LIN {X -0.121,Y -401.497,Z 1324.427,A 0.000,B 0.000,C 90.000,E1 292.823} C_DIS
LIN {X 0.045,Y -401.770,Z 1324.423,A 0.000,B 0.000,C 90.000,E1 292.099} C_DIS
LIN {X 0.005,Y -404.574,Z 1324.396,A 0.000,B 0.000,C 90.000,E1 287.221} C_DIS
LIN {X 0.106,Y -404.760,Z 1324.394,A 0.000,B 0.000,C 90.000,E1 286.858} C_DIS
LIN {X 0.013,Y -406.044,Z 1324.365,A 0.000,B 0.000,C 90.000,E1 281.658} C_DIS
LIN {X 0.103,Y -406.134,Z 1324.363,A 0.000,B 0.000,C 90.000,E1 281.299} C_DIS
LIN {X 0.132,Y -405.657,Z 1324.334,A 0.000,B 0.000,C 90.000,E1 276.087} C_DIS
LIN {X 0.138,Y -405.595,Z 1324.332,A 0.000,B 0.000,C 90.000,E1 275.739} C_DIS
LIN {X -0.193,Y -403.547,Z 1324.305,A 0.000,B 0.000,C 90.000,E1 270.917} C_DIS
LIN {X 0.146,Y -403.030,Z 1324.301,A 0.000,B 0.000,C 90.000,E1 270.172} C_DIS
LIN {X -0.032,Y -399.006,Z 1324.272,A 0.000,B 0.000,C 90.000,E1 264.951} C_DIS
LIN {X -0.006,Y -395.117,Z 1324.254,A 0.000,B 0.000,C 90.000,E1 261.781} C_DIS
LIN {X 0.129,Y -392.916,Z 1324.241,A 0.000,B 0.000,C 90.000,E1 259.285} C_DIS
LIN {X 0.120,Y -391.854,Z 1324.237,A 0.000,B 0.000,C 90.000,E1 258.578} C_DIS
LIN {X -0.125,Y -385.723,Z 1324.211,A 0.000,B 0.000,C 90.000,E1 253.976} C_DIS
LIN {X -0.189,Y -384.951,Z 1324.207,A 0.000,B 0.000,C 90.000,E1 253.268} C_DIS
LIN {X 0.038,Y -378.101,Z 1324.183,A 0.000,B 0.000,C 90.000,E1 248.901} C_DIS
LIN {X -0.226,Y -376.344,Z 1324.175,A 0.000,B 0.000,C 90.000,E1 247.486} C_DIS
LIN {X -0.100,Y -375.834,Z 1324.173,A 0.000,B 0.000,C 90.000,E1 247.102} C_DIS
LIN {X 0.018,Y -369.070,Z 1324.150,A 0.000,B 0.000,C 90.000,E1 243.050} C_DIS
LIN {X -0.071,Y -366.221,Z 1324.138,A 0.000,B 0.000,C 90.000,E1 240.845} C_DIS
LIN {X 0.090,Y -358.817,Z 1324.113,A 0.000,B 0.000,C 90.000,E1 236.342} C_DIS
LIN {X -0.119,Y -356.008,Z 1324.101,A 0.000,B 0.000,C 90.000,E1 234.116} C_DIS
LIN {X -0.138,Y -350.728,Z 1324.083,A 0.000,B 0.000,C 90.000,E1 230.884} C_DIS
LIN {X -0.156,Y -350.742,Z 1324.083,A 0.000,B 0.000,C 90.000,E1 230.884} C_DIS
LIN {X 0.060,Y -364.108,Z 1324.069,A 0.000,B 0.000,C 90.000,E1 228.405} C_DIS
LIN {X -0.264,Y -378.946,Z 1324.056,A 0.000,B 0.000,C 90.000,E1 226.053} C_DIS
LIN {X -0.195,Y -395.284,Z 1324.043,A 0.000,B 0.000,C 90.000,E1 223.704} C_DIS
LIN {X -0.073,Y -413.058,Z 1324.030,A 0.000,B 0.000,C 90.000,E1 221.434} C_DIS
LIN {X -0.030,Y -432.976,Z 1324.018,A 0.000,B 0.000,C 90.000,E1 219.197} C_DIS
LIN {X -0.195,Y -443.092,Z 1324.012,A 0.000,B 0.000,C 90.000,E1 218.177} C_DIS
LIN {X -0.039,Y -444.761,Z 1324.010,A 0.000,B 0.000,C 90.000,E1 217.855} C_DIS
LIN {X -0.002,Y -445.959,Z 1324.009,A 0.000,B 0.000,C 90.000,E1 217.523} C_DIS
LIN {X -0.039,Y -446.904,Z 1324.007,A 0.000,B 0.000,C 90.000,E1 217.202} C_DIS
LIN {X 0.012,Y -447.701,Z 1324.005,A 0.000,B 0.000,C 90.000,E1 216.870} C_DIS
LIN {X 0.036,Y -448.929,Z 1324.001,A 0.000,B 0.000,C 90.000,E1 216.217} C_DIS
LIN {X -0.193,Y -449.875,Z 1323.998,A 0.000,B 0.000,C 90.000,E1 215.598} C_DIS
LIN {X -0.078,Y -450.866,Z 1323.992,A 0.000,B 0.000,C 90.000,E1 214.612} C_DIS
LIN {X 0.114,Y -453.547,Z 1323.978,A 0.000,B 0.000,C 90.000,E1 212.005} C_DIS
LIN {X -0.202,Y -456.066,Z 1323.965,A 0.000,B 0.000,C 90.000,E1 209.795} C_DIS
LIN {X 0.116,Y -458.841,Z 1323.953,A 0.000,B 0.000,C 90.000,E1 207.513} C_DIS
LIN {X 0.098,Y -462.041,Z 1323.941,A 0.000,B 0.000,C 90.000,E1 205.283} C_DIS
LIN {X -0.010,Y -463.926,Z 1323.933,A 0.000,B 0.000,C 90.000,E1 204.027} C_DIS
LIN {X -0.094,Y -465.699,Z 1323.927,A 0.000,B 0.000,C 90.000,E1 202.770} C_DIS
LIN {X 0.048,Y -467.836,Z 1323.918,A 0.000,B 0.000,C 90.000,E1 201.173} C_DIS
LIN {X 0.137,Y -470.708,Z 1323.906,A 0.000,B 0.000,C 90.000,E1 198.960} C_DIS
LIN {X 0.019,Y -473.212,Z 1323.895,A 0.000,B 0.000,C 90.000,E1 197.094} C_DIS
LIN {X -0.181,Y -475.587,Z 1323.885,A 0.000,B 0.000,C 90.000,E1 195.245} C_DIS
LIN {X 0.009,Y -477.937,Z 1323.874,A 0.000,B 0.000,C 90.000,E1 193.355} C_DIS
LIN {X 0.002,Y -480.638,Z 1323.862,A 0.000,B 0.000,C 90.000,E1 191.186} C_DIS
LIN {X 0.243,Y -482.542,Z 1323.854,A 0.000,B 0.000,C 90.000,E1 189.613} C_DIS
LIN {X -0.036,Y -484.416,Z 1323.845,A 0.000,B 0.000,C 90.000,E1 188.106} C_DIS
LIN {X 0.139,Y -486.155,Z 1323.837,A 0.000,B 0.000,C 90.000,E1 186.549} C_DIS
LIN {X 0.040,Y -487.423,Z 1323.830,A 0.000,B 0.000,C 90.000,E1 185.334} C_DIS
LIN {X 0.053,Y -489.054,Z 1323.819,A 0.000,B 0.000,C 90.000,E1 183.498} C_DIS
LIN {X -0.246,Y -490.104,Z 1323.811,A 0.000,B 0.000,C 90.000,E1 182.007} C_DIS
LIN {X -0.041,Y -490.805,Z 1323.803,A 0.000,B 0.000,C 90.000,E1 180.458} C_DIS
LIN {X 0.166,Y -491.124,Z 1323.794,A 0.000,B 0.000,C 90.000,E1 178.912} C_DIS
LIN {X -0.145,Y -491.170,Z 1323.791,A 0.000,B 0.000,C 90.000,E1 178.339} C_DIS
LIN {X 0.097,Y -490.879,Z 1323.782,A 0.000,B 0.000,C 90.000,E1 176.788} C_DIS
LIN {X -0.019,Y -490.174,Z 1323.776,A 0.000,B 0.000,C 90.000,E1 175.584} C_DIS
LIN {X 0.012,Y -489.462,Z 1323.770,A 0.000,B 0.000,C 90.000,E1 174.666} C_DIS
LIN {X 0.080,Y -488.430,Z 1323.765,A 0.000,B 0.000,C 90.000,E1 173.742} C_DIS
LIN {X -0.221,Y -487.716,Z 1323.762,A 0.000,B 0.000,C 90.000,E1 173.166} C_DIS
LIN {X -0.046,Y -486.853,Z 1323.759,A 0.000,B 0.000,C 90.000,E1 172.534} C_DIS
LIN {X 0.061,Y -485.258,Z 1323.753,A 0.000,B 0.000,C 90.000,E1 171.602} C_DIS
LIN {X 0.081,Y -483.312,Z 1323.748,A 0.000,B 0.000,C 90.000,E1 170.679} C_DIS
LIN {X 0.155,Y -481.094,Z 1323.743,A 0.000,B 0.000,C 90.000,E1 169.746} C_DIS
LIN {X 0.204,Y -478.140,Z 1323.738,A 0.000,B 0.000,C 90.000,E1 168.814} C_DIS
LIN {X -0.094,Y -475.795,Z 1323.735,A 0.000,B 0.000,C 90.000,E1 168.229} C_DIS
LIN {X -0.010,Y -471.370,Z 1323.729,A 0.000,B 0.000,C 90.000,E1 167.285} C_DIS
LIN {X -0.087,Y -465.612,Z 1323.724,A 0.000,B 0.000,C 90.000,E1 166.353} C_DIS
LIN {X 0.163,Y -454.836,Z 1323.714,A 0.000,B 0.000,C 90.000,E1 164.574} C_DIS
LIN {X 0.161,Y -445.144,Z 1323.705,A 0.000,B 0.000,C 90.000,E1 162.960} C_DIS
LIN {X 0.148,Y -439.297,Z 1323.699,A 0.000,B 0.000,C 90.000,E1 161.819} C_DIS
LIN {X -0.145,Y -437.494,Z 1323.696,A 0.000,B 0.000,C 90.000,E1 161.221} C_DIS
LIN {X 0.105,Y -436.906,Z 1323.694,A 0.000,B 0.000,C 90.000,E1 160.859} C_DIS
LIN {X -0.061,Y -436.819,Z 1323.692,A 0.000,B 0.000,C 90.000,E1 160.550} C_DIS
LIN {X 0.013,Y -438.051,Z 1323.690,A 0.000,B 0.000,C 90.000,E1 160.134} C_DIS
LIN {X 0.121,Y -438.069,Z 1323.690,A 0.000,B 0.000,C 90.000,E1 160.115} C_DIS
LIN {X 0.145,Y -440.213,Z 1323.688,A 0.000,B 0.000,C 90.000,E1 159.880} C_DIS
LIN {X -0.083,Y -441.492,Z 1323.688,A 0.000,B 0.000,C 90.000,E1 159.752} C_DIS
LIN {X 0.103,Y -450.346,Z 1323.683,A 0.000,B 0.000,C 90.000,E1 158.975} C_DIS
LIN {X 0.249,Y -462.852,Z 1323.678,A 0.000,B 0.000,C 90.000,E1 157.975} C_DIS
LIN {X -0.095,Y -473.715,Z 1323.673,A 0.000,B 0.000,C 90.000,E1 157.177} C_DIS
LIN {X 0.021,Y -484.245,Z 1323.668,A 0.000,B 0.000,C 90.000,E1 156.305} C_DIS
LIN {X 0.027,Y -491.350,Z 1323.665,A 0.000,B 0.000,C 90.000,E1 155.665} C_DIS
LIN {X 0.255,Y -498.290,Z 1323.661,A 0.000,B 0.000,C 90.000,E1 154.973} C_DIS
LIN {X 0.202,Y -506.494,Z 1323.657,A 0.000,B 0.000,C 90.000,E1 154.152} C_DIS
LIN {X -0.144,Y -514.176,Z 1323.652,A 0.000,B 0.000,C 90.000,E1 153.332} C_DIS
LIN {X 0.066,Y -517.855,Z 1323.649,A 0.000,B 0.000,C 90.000,E1 152.871} C_DIS
LIN {X -0.273,Y -520.234,Z 1323.648,A 0.000,B 0.000,C 90.000,E1 152.615} C_DIS
LIN {X -0.226,Y -524.431,Z 1323.645,A 0.000,B 0.000,C 90.000,E1 152.025} C_DIS
LIN {X 0.162,Y -528.939,Z 1323.641,A 0.000,B 0.000,C 90.000,E1 151.257} C_DIS
LIN {X -0.186,Y -531.948,Z 1323.637,A 0.000,B 0.000,C 90.000,E1 150.717} C_DIS
LIN {X -0.048,Y -534.414,Z 1323.634,A 0.000,B 0.000,C 90.000,E1 150.127} C_DIS
LIN {X 0.106,Y -536.377,Z 1323.631,A 0.000,B 0.000,C 90.000,E1 149.537} C_DIS
LIN {X -0.190,Y -538.148,Z 1323.628,A 0.000,B 0.000,C 90.000,E1 148.997} C_DIS
LIN {X -0.013,Y -539.691,Z 1323.625,A 0.000,B 0.000,C 90.000,E1 148.408} C_DIS
LIN {X 0.183,Y -541.656,Z 1323.620,A 0.000,B 0.000,C 90.000,E1 147.533} C_DIS
LIN {X -0.077,Y -542.760,Z 1323.617,A 0.000,B 0.000,C 90.000,E1 146.993} C_DIS
LIN {X -0.003,Y -544.135,Z 1323.612,A 0.000,B 0.000,C 90.000,E1 146.135} C_DIS
LIN {X -0.212,Y -545.265,Z 1323.607,A 0.000,B 0.000,C 90.000,E1 145.308} C_DIS
LIN {X 0.349,Y -546.179,Z 1323.603,A 0.000,B 0.000,C 90.000,E1 144.402} C_DIS
LIN {X -0.243,Y -547.175,Z 1323.596,A 0.000,B 0.000,C 90.000,E1 143.336} C_DIS
LIN {X 0.086,Y -548.739,Z 1323.585,A 0.000,B 0.000,C 90.000,E1 141.331} C_DIS
LIN {X -0.243,Y -549.253,Z 1323.582,A 0.000,B 0.000,C 90.000,E1 140.803} C_DIS
LIN {X -0.163,Y -549.755,Z 1323.581,A 0.000,B 0.000,C 90.000,E1 140.517} C_DIS
LIN {X -0.030,Y -550.405,Z 1323.579,A 0.000,B 0.000,C 90.000,E1 140.275} C_DIS
LIN {X -0.098,Y -550.908,Z 1323.579,A 0.000,B 0.000,C 90.000,E1 140.194} C_DIS
LIN {X -0.011,Y -551.251,Z 1323.579,A 0.000,B 0.000,C 90.000,E1 140.150} C_DIS
LIN {X 0.193,Y -553.747,Z 1323.578,A 0.000,B 0.000,C 90.000,E1 139.989} C_DIS
LIN {X -0.092,Y -561.011,Z 1323.577,A 0.000,B 0.000,C 90.000,E1 139.784} C_DIS
LIN {X -0.058,Y -566.314,Z 1323.576,A 0.000,B 0.000,C 90.000,E1 139.622} C_DIS
LIN {X 0.041,Y -572.536,Z 1323.574,A 0.000,B 0.000,C 90.000,E1 139.380} C_DIS
LIN {X 0.025,Y -575.274,Z 1323.574,A 0.000,B 0.000,C 90.000,E1 139.256} C_DIS
LIN {X 0.100,Y -578.139,Z 1323.573,A 0.000,B 0.000,C 90.000,E1 139.094} C_DIS
LIN {X 0.102,Y -583.931,Z 1323.571,A 0.000,B 0.000,C 90.000,E1 138.728} C_DIS
LIN {X 0.179,Y -589.629,Z 1323.569,A 0.000,B 0.000,C 90.000,E1 138.324} C_DIS
LIN {X -0.289,Y -592.300,Z 1323.568,A 0.000,B 0.000,C 90.000,E1 138.162} C_DIS
LIN {X -0.249,Y -597.402,Z 1323.565,A 0.000,B 0.000,C 90.000,E1 137.715} C_DIS
LIN {X 0.026,Y -603.693,Z 1323.562,A 0.000,B 0.000,C 90.000,E1 137.067} C_DIS
LIN {X 0.039,Y -609.589,Z 1323.558,A 0.000,B 0.000,C 90.000,E1 136.419} C_DIS
LIN {X -0.392,Y -614.960,Z 1323.554,A 0.000,B 0.000,C 90.000,E1 135.810} C_DIS
LIN {X 0.074,Y -619.928,Z 1323.551,A 0.000,B 0.000,C 90.000,E1 135.121} C_DIS
LIN {X 0.077,Y -625.397,Z 1323.547,A 0.000,B 0.000,C 90.000,E1 134.352} C_DIS
LIN {X 0.197,Y -629.756,Z 1323.543,A 0.000,B 0.000,C 90.000,E1 133.704} C_DIS
LIN {X 0.205,Y -636.392,Z 1323.537,A 0.000,B 0.000,C 90.000,E1 132.690} C_DIS
LIN {X -0.139,Y -644.193,Z 1323.530,A 0.000,B 0.000,C 90.000,E1 131.472} C_DIS
LIN {X -0.369,Y -649.561,Z 1323.526,A 0.000,B 0.000,C 90.000,E1 130.620} C_DIS
LIN {X 0.390,Y -655.307,Z 1323.520,A 0.000,B 0.000,C 90.000,E1 129.564} C_DIS
LIN {X -0.142,Y -660.174,Z 1323.515,A 0.000,B 0.000,C 90.000,E1 128.749} C_DIS
LIN {X 0.444,Y -665.225,Z 1323.510,A 0.000,B 0.000,C 90.000,E1 127.729} C_DIS
LIN {X 0.033,Y -668.149,Z 1323.506,A 0.000,B 0.000,C 90.000,E1 127.156} C_DIS
LIN {X 0.098,Y -671.391,Z 1323.502,A 0.000,B 0.000,C 90.000,E1 126.423} C_DIS
LIN {X -0.208,Y -674.346,Z 1323.498,A 0.000,B 0.000,C 90.000,E1 125.724} C_DIS
LIN {X 0.070,Y -677.016,Z 1323.494,A 0.000,B 0.000,C 90.000,E1 124.978} C_DIS
LIN {X -0.177,Y -679.417,Z 1323.490,A 0.000,B 0.000,C 90.000,E1 124.278} C_DIS
LIN {X 0.155,Y -682.105,Z 1323.485,A 0.000,B 0.000,C 90.000,E1 123.293} C_DIS
LIN {X -0.056,Y -683.932,Z 1323.481,A 0.000,B 0.000,C 90.000,E1 122.594} C_DIS
LIN {X -0.414,Y -686.028,Z 1323.476,A 0.000,B 0.000,C 90.000,E1 121.671} C_DIS
LIN {X 0.207,Y -687.810,Z 1323.471,A 0.000,B 0.000,C 90.000,E1 120.669} C_DIS
LIN {X -0.316,Y -688.916,Z 1323.467,A 0.000,B 0.000,C 90.000,E1 120.001} C_DIS
LIN {X -0.231,Y -689.846,Z 1323.463,A 0.000,B 0.000,C 90.000,E1 119.283} C_DIS
LIN {X -0.270,Y -690.650,Z 1323.456,A 0.000,B 0.000,C 90.000,E1 118.103} C_DIS
LIN {X 0.070,Y -690.922,Z 1323.451,A 0.000,B 0.000,C 90.000,E1 117.129} C_DIS
LIN {X 0.102,Y -690.918,Z 1323.446,A 0.000,B 0.000,C 90.000,E1 116.181} C_DIS
LIN {X 0.197,Y -690.516,Z 1323.442,A 0.000,B 0.000,C 90.000,E1 115.463} C_DIS
LIN {X -0.247,Y -690.085,Z 1323.439,A 0.000,B 0.000,C 90.000,E1 115.027} C_DIS
LIN {X 0.222,Y -689.384,Z 1323.436,A 0.000,B 0.000,C 90.000,E1 114.515} C_DIS
LIN {X -0.226,Y -688.116,Z 1323.434,A 0.000,B 0.000,C 90.000,E1 114.079} C_DIS
LIN {X 0.002,Y -687.201,Z 1323.432,A 0.000,B 0.000,C 90.000,E1 113.823} C_DIS
LIN {X 0.173,Y -684.800,Z 1323.430,A 0.000,B 0.000,C 90.000,E1 113.334} C_DIS
LIN {X 0.281,Y -683.875,Z 1323.429,A 0.000,B 0.000,C 90.000,E1 113.206} C_DIS
LIN {X -0.205,Y -680.137,Z 1323.427,A 0.000,B 0.000,C 90.000,E1 112.898} C_DIS
LIN {X -0.053,Y -677.976,Z 1323.426,A 0.000,B 0.000,C 90.000,E1 112.695} C_DIS
LIN {X -0.130,Y -675.714,Z 1323.426,A 0.000,B 0.000,C 90.000,E1 112.589} C_DIS
LIN {X -0.167,Y -667.939,Z 1323.424,A 0.000,B 0.000,C 90.000,E1 112.280} C_DIS
LIN {X -0.136,Y -665.627,Z 1323.423,A 0.000,B 0.000,C 90.000,E1 112.206} C_DIS
LIN {X 0.045,Y -656.434,Z 1323.422,A 0.000,B 0.000,C 90.000,E1 112.025} C_DIS
LIN {X 0.092,Y -645.125,Z 1323.422,A 0.000,B 0.000,C 90.000,E1 111.897} C_DIS
LIN {X -0.126,Y -643.838,Z 1323.422,A 0.000,B 0.000,C 90.000,E1 111.897} C_DIS
LIN {X -0.123,Y -642.190,Z 1323.421,A 0.000,B 0.000,C 90.000,E1 111.844} C_DIS
LIN {X -0.163,Y -642.114,Z 1323.421,A 0.000,B 0.000,C 90.000,E1 111.844} C_DIS
LIN {X -0.157,Y -643.175,Z 1323.420,A 0.000,B 0.000,C 90.000,E1 111.642} C_DIS
LIN {X 0.366,Y -648.272,Z 1323.417,A 0.000,B 0.000,C 90.000,E1 110.972} C_DIS
LIN {X 0.249,Y -651.211,Z 1323.415,A 0.000,B 0.000,C 90.000,E1 110.610} C_DIS
LIN {X 0.056,Y -656.148,Z 1323.411,A 0.000,B 0.000,C 90.000,E1 109.885} C_DIS
LIN {X 0.080,Y -659.795,Z 1323.407,A 0.000,B 0.000,C 90.000,E1 109.268} C_DIS
LIN {X -0.030,Y -663.395,Z 1323.403,A 0.000,B 0.000,C 90.000,E1 108.544} C_DIS
LIN {X -0.112,Y -666.500,Z 1323.399,A 0.000,B 0.000,C 90.000,E1 107.819} C_DIS
LIN {X -0.084,Y -668.382,Z 1323.396,A 0.000,B 0.000,C 90.000,E1 107.330} C_DIS
LIN {X -0.317,Y -670.917,Z 1323.392,A 0.000,B 0.000,C 90.000,E1 106.622} C_DIS
LIN {X -0.267,Y -672.413,Z 1323.390,A 0.000,B 0.000,C 90.000,E1 106.134} C_DIS
LIN {X 0.194,Y -674.333,Z 1323.385,A 0.000,B 0.000,C 90.000,E1 105.371} C_DIS
LIN {X 0.033,Y -675.890,Z 1323.381,A 0.000,B 0.000,C 90.000,E1 104.662} C_DIS
LIN {X 0.099,Y -676.838,Z 1323.379,A 0.000,B 0.000,C 90.000,E1 104.175} C_DIS
LIN {X 0.003,Y -677.587,Z 1323.376,A 0.000,B 0.000,C 90.000,E1 103.703} C_DIS
LIN {X -0.245,Y -678.142,Z 1323.374,A 0.000,B 0.000,C 90.000,E1 103.244} C_DIS
LIN {X 0.290,Y -678.596,Z 1323.370,A 0.000,B 0.000,C 90.000,E1 102.479} C_DIS
LIN {X 0.206,Y -678.770,Z 1323.367,A 0.000,B 0.000,C 90.000,E1 102.007} C_DIS
LIN {X 0.075,Y -678.561,Z 1323.363,A 0.000,B 0.000,C 90.000,E1 101.299} C_DIS
LIN {X -0.145,Y -678.203,Z 1323.360,A 0.000,B 0.000,C 90.000,E1 100.838} C_DIS
LIN {X -0.239,Y -677.602,Z 1323.358,A 0.000,B 0.000,C 90.000,E1 100.366} C_DIS
LIN {X 0.208,Y -676.798,Z 1323.355,A 0.000,B 0.000,C 90.000,E1 99.849} C_DIS
LIN {X 0.099,Y -675.724,Z 1323.352,A 0.000,B 0.000,C 90.000,E1 99.378} C_DIS
LIN {X -0.068,Y -675.093,Z 1323.351,A 0.000,B 0.000,C 90.000,E1 99.151} C_DIS
LIN {X -0.193,Y -673.531,Z 1323.348,A 0.000,B 0.000,C 90.000,E1 98.681} C_DIS
LIN {X 0.234,Y -671.646,Z 1323.345,A 0.000,B 0.000,C 90.000,E1 98.163} C_DIS
LIN {X -0.014,Y -669.538,Z 1323.343,A 0.000,B 0.000,C 90.000,E1 97.701} C_DIS
LIN {X 0.297,Y -665.986,Z 1323.339,A 0.000,B 0.000,C 90.000,E1 96.947} C_DIS
LIN {X 0.010,Y -663.432,Z 1323.336,A 0.000,B 0.000,C 90.000,E1 96.486} C_DIS
LIN {X 0.174,Y -659.143,Z 1323.332,A 0.000,B 0.000,C 90.000,E1 95.739} C_DIS
LIN {X -0.153,Y -656.013,Z 1323.329,A 0.000,B 0.000,C 90.000,E1 95.277} C_DIS
LIN {X 0.196,Y -653.522,Z 1323.327,A 0.000,B 0.000,C 90.000,E1 94.878} C_DIS
LIN {X -0.271,Y -648.929,Z 1323.324,A 0.000,B 0.000,C 90.000,E1 94.302} C_DIS
LIN {X -0.018,Y -645.076,Z 1323.321,A 0.000,B 0.000,C 90.000,E1 93.784} C_DIS
LIN {X 0.164,Y -640.881,Z 1323.318,A 0.000,B 0.000,C 90.000,E1 93.269} C_DIS
LIN {X 0.229,Y -635.195,Z 1323.315,A 0.000,B 0.000,C 90.000,E1 92.636} C_DIS
LIN {X 0.278,Y -629.016,Z 1323.311,A 0.000,B 0.000,C 90.000,E1 92.007} C_DIS
LIN {X -0.068,Y -623.989,Z 1323.309,A 0.000,B 0.000,C 90.000,E1 91.547} C_DIS
LIN {X -0.154,Y -617.687,Z 1323.305,A 0.000,B 0.000,C 90.000,E1 90.974} C_DIS
LIN {X -0.212,Y -616.327,Z 1323.305,A 0.000,B 0.000,C 90.000,E1 90.859} C_DIS
LIN {X -0.119,Y -608.933,Z 1323.302,A 0.000,B 0.000,C 90.000,E1 90.286} C_DIS
LIN {X 0.022,Y -602.442,Z 1323.299,A 0.000,B 0.000,C 90.000,E1 89.885} C_DIS
LIN {X -0.005,Y -595.811,Z 1323.297,A 0.000,B 0.000,C 90.000,E1 89.542} C_DIS
LIN {X -0.209,Y -588.759,Z 1323.296,A 0.000,B 0.000,C 90.000,E1 89.255} C_DIS
LIN {X -0.279,Y -576.942,Z 1323.293,A 0.000,B 0.000,C 90.000,E1 88.797} C_DIS
LIN {X 0.047,Y -574.599,Z 1323.292,A 0.000,B 0.000,C 90.000,E1 88.625} C_DIS
LIN {X 0.007,Y -573.046,Z 1323.292,A 0.000,B 0.000,C 90.000,E1 88.511} C_DIS
LIN {X -0.222,Y -572.379,Z 1323.291,A 0.000,B 0.000,C 90.000,E1 88.453} C_DIS
LIN {X -0.265,Y -572.358,Z 1323.291,A 0.000,B 0.000,C 90.000,E1 88.453} C_DIS
LIN {X 0.105,Y -571.730,Z 1323.290,A 0.000,B 0.000,C 90.000,E1 88.165} C_DIS
LIN {X 0.242,Y -571.611,Z 1323.288,A 0.000,B 0.000,C 90.000,E1 87.879} C_DIS
LIN {X -0.194,Y -571.647,Z 1323.287,A 0.000,B 0.000,C 90.000,E1 87.650} C_DIS
LIN {X -0.017,Y -573.901,Z 1323.273,A 0.000,B 0.000,C 90.000,E1 85.179} C_DIS
LIN {X 0.281,Y -576.662,Z 1323.260,A 0.000,B 0.000,C 90.000,E1 82.704} C_DIS
LIN {X 0.020,Y -578.299,Z 1323.252,A 0.000,B 0.000,C 90.000,E1 81.376} C_DIS
LIN {X -0.249,Y -580.537,Z 1323.242,A 0.000,B 0.000,C 90.000,E1 79.511} C_DIS
LIN {X -0.019,Y -581.688,Z 1323.236,A 0.000,B 0.000,C 90.000,E1 78.409} C_DIS
LIN {X 0.001,Y -582.953,Z 1323.228,A 0.000,B 0.000,C 90.000,E1 77.061} C_DIS
LIN {X -0.151,Y -584.243,Z 1323.219,A 0.000,B 0.000,C 90.000,E1 75.463} C_DIS
LIN {X -0.114,Y -585.343,Z 1323.210,A 0.000,B 0.000,C 90.000,E1 73.850} C_DIS
LIN {X 0.102,Y -586.253,Z 1323.203,A 0.000,B 0.000,C 90.000,E1 72.489} C_DIS
LIN {X -0.205,Y -587.317,Z 1323.194,A 0.000,B 0.000,C 90.000,E1 70.913} C_DIS
LIN {X 0.268,Y -588.225,Z 1323.185,A 0.000,B 0.000,C 90.000,E1 69.263} C_DIS
LIN {X -0.219,Y -589.154,Z 1323.178,A 0.000,B 0.000,C 90.000,E1 67.975} C_DIS
LIN {X 0.071,Y -590.026,Z 1323.170,A 0.000,B 0.000,C 90.000,E1 66.613} C_DIS
LIN {X -0.028,Y -591.140,Z 1323.161,A 0.000,B 0.000,C 90.000,E1 65.025} C_DIS
LIN {X -0.190,Y -592.477,Z 1323.151,A 0.000,B 0.000,C 90.000,E1 63.179} C_DIS
LIN {X -0.153,Y -594.247,Z 1323.139,A 0.000,B 0.000,C 90.000,E1 61.051} C_DIS
LIN {X -0.007,Y -596.300,Z 1323.127,A 0.000,B 0.000,C 90.000,E1 58.918} C_DIS
LIN {X 0.283,Y -598.201,Z 1323.117,A 0.000,B 0.000,C 90.000,E1 57.041} C_DIS
LIN {X 0.194,Y -599.896,Z 1323.108,A 0.000,B 0.000,C 90.000,E1 55.468} C_DIS
LIN {X -0.262,Y -601.231,Z 1323.101,A 0.000,B 0.000,C 90.000,E1 54.196} C_DIS
LIN {X -0.081,Y -602.650,Z 1323.092,A 0.000,B 0.000,C 90.000,E1 52.603} C_DIS
LIN {X 0.094,Y -603.521,Z 1323.086,A 0.000,B 0.000,C 90.000,E1 51.537} C_DIS
LIN {X -0.155,Y -604.572,Z 1323.078,A 0.000,B 0.000,C 90.000,E1 49.989} C_DIS
LIN {X 0.151,Y -605.035,Z 1323.073,A 0.000,B 0.000,C 90.000,E1 49.175} C_DIS
LIN {X -0.195,Y -605.390,Z 1323.068,A 0.000,B 0.000,C 90.000,E1 48.162} C_DIS
LIN {X -0.089,Y -605.535,Z 1323.062,A 0.000,B 0.000,C 90.000,E1 47.106} C_DIS
LIN {X -0.205,Y -605.737,Z 1323.054,A 0.000,B 0.000,C 90.000,E1 45.810} C_DIS
LIN {X 0.075,Y -605.733,Z 1323.050,A 0.000,B 0.000,C 90.000,E1 45.000} C_DIS
LIN {X 0.355,Y -605.614,Z 1323.046,A 0.000,B 0.000,C 90.000,E1 44.190} C_DIS
LIN {X -0.175,Y -605.174,Z 1323.038,A 0.000,B 0.000,C 90.000,E1 42.933} C_DIS
LIN {X 0.340,Y -604.882,Z 1323.033,A 0.000,B 0.000,C 90.000,E1 41.838} C_DIS
LIN {X 0.040,Y -604.252,Z 1323.024,A 0.000,B 0.000,C 90.000,E1 40.297} C_DIS
LIN {X 0.006,Y -603.596,Z 1323.017,A 0.000,B 0.000,C 90.000,E1 38.991} C_DIS
LIN {X 0.306,Y -603.209,Z 1323.012,A 0.000,B 0.000,C 90.000,E1 38.177} C_DIS
LIN {X -0.248,Y -602.675,Z 1323.008,A 0.000,B 0.000,C 90.000,E1 37.443} C_DIS
LIN {X -0.075,Y -601.551,Z 1323.002,A 0.000,B 0.000,C 90.000,E1 36.377} C_DIS
LIN {X -0.165,Y -600.463,Z 1322.998,A 0.000,B 0.000,C 90.000,E1 35.598} C_DIS
LIN {X -0.127,Y -598.272,Z 1322.990,A 0.000,B 0.000,C 90.000,E1 34.278} C_DIS
LIN {X -0.028,Y -596.179,Z 1322.984,A 0.000,B 0.000,C 90.000,E1 33.214} C_DIS
LIN {X -0.009,Y -594.349,Z 1322.980,A 0.000,B 0.000,C 90.000,E1 32.418} C_DIS
LIN {X 0.310,Y -592.267,Z 1322.976,A 0.000,B 0.000,C 90.000,E1 31.592} C_DIS
LIN {X 0.294,Y -589.804,Z 1322.971,A 0.000,B 0.000,C 90.000,E1 30.797} C_DIS
LIN {X 0.256,Y -587.127,Z 1322.967,A 0.000,B 0.000,C 90.000,E1 30.001} C_DIS
LIN {X 0.188,Y -583.925,Z 1322.962,A 0.000,B 0.000,C 90.000,E1 29.205} C_DIS
LIN {X -0.128,Y -581.034,Z 1322.959,A 0.000,B 0.000,C 90.000,E1 28.565} C_DIS
LIN {X -0.193,Y -577.785,Z 1322.955,A 0.000,B 0.000,C 90.000,E1 27.897} C_DIS
LIN {X 0.028,Y -575.022,Z 1322.952,A 0.000,B 0.000,C 90.000,E1 27.334} C_DIS
LIN {X -0.100,Y -571.222,Z 1322.948,A 0.000,B 0.000,C 90.000,E1 26.668} C_DIS
LIN {X -0.008,Y -567.147,Z 1322.944,A 0.000,B 0.000,C 90.000,E1 25.976} C_DIS
LIN {X 0.048,Y -562.716,Z 1322.941,A 0.000,B 0.000,C 90.000,E1 25.283} C_DIS
LIN {X -0.205,Y -559.084,Z 1322.938,A 0.000,B 0.000,C 90.000,E1 24.771} C_DIS
LIN {X 0.205,Y -551.871,Z 1322.932,A 0.000,B 0.000,C 90.000,E1 23.770} C_DIS
LIN {X 0.124,Y -546.219,Z 1322.928,A 0.000,B 0.000,C 90.000,E1 23.078} C_DIS
LIN {X -0.116,Y -536.469,Z 1322.922,A 0.000,B 0.000,C 90.000,E1 21.972} C_DIS
LIN {X -0.014,Y -532.645,Z 1322.920,A 0.000,B 0.000,C 90.000,E1 21.535} C_DIS
LIN {X 0.033,Y -522.333,Z 1322.914,A 0.000,B 0.000,C 90.000,E1 20.429} C_DIS
LIN {X 0.089,Y -513.120,Z 1322.908,A 0.000,B 0.000,C 90.000,E1 19.450} C_DIS
LIN {X 0.175,Y -502.525,Z 1322.902,A 0.000,B 0.000,C 90.000,E1 18.362} C_DIS
LIN {X -0.160,Y -492.885,Z 1322.897,A 0.000,B 0.000,C 90.000,E1 17.457} C_DIS
LIN {X 0.206,Y -483.354,Z 1322.892,A 0.000,B 0.000,C 90.000,E1 16.496} C_DIS
LIN {X 0.158,Y -473.255,Z 1322.887,A 0.000,B 0.000,C 90.000,E1 15.552} C_DIS
LIN {X -0.205,Y -458.586,Z 1322.879,A 0.000,B 0.000,C 90.000,E1 14.245} C_DIS
LIN {X 0.034,Y -435.463,Z 1322.866,A 0.000,B 0.000,C 90.000,E1 11.951} C_DIS
LIN {X -0.074,Y -418.356,Z 1322.856,A 0.000,B 0.000,C 90.000,E1 10.141} C_DIS
LIN {X 0.053,Y -402.790,Z 1322.847,A 0.000,B 0.000,C 90.000,E1 8.398} C_DIS
LIN {X -0.107,Y -398.609,Z 1322.844,A 0.000,B 0.000,C 90.000,E1 7.936} C_DIS
LIN {X -0.059,Y -395.385,Z 1322.841,A 0.000,B 0.000,C 90.000,E1 7.466} C_DIS
LIN {X -0.097,Y -395.367,Z 1322.841,A 0.000,B 0.000,C 90.000,E1 7.466} C_DIS
LIN {X 0.017,Y -395.978,Z 1322.841,A 0.000,B 0.000,C 90.000,E1 7.296} C_DIS
LIN {X -0.022,Y -396.010,Z 1322.841,A 0.000,B 0.000,C 90.000,E1 7.296} C_DIS
LIN {X -0.068,Y -399.318,Z 1322.839,A 0.000,B 0.000,C 90.000,E1 7.004} C_DIS
LIN {X -0.013,Y -404.877,Z 1322.837,A 0.000,B 0.000,C 90.000,E1 6.606} C_DIS
LIN {X 0.149,Y -412.803,Z 1322.834,A 0.000,B 0.000,C 90.000,E1 6.087} C_DIS
LIN {X -0.157,Y -416.164,Z 1322.833,A 0.000,B 0.000,C 90.000,E1 5.910} C_DIS
LIN {X -0.099,Y -423.981,Z 1322.830,A 0.000,B 0.000,C 90.000,E1 5.334} C_DIS
LIN {X 0.170,Y -428.633,Z 1322.828,A 0.000,B 0.000,C 90.000,E1 4.935} C_DIS
LIN {X -0.042,Y -437.502,Z 1322.823,A 0.000,B 0.000,C 90.000,E1 4.188} C_DIS
LIN {X -0.075,Y -442.014,Z 1322.821,A 0.000,B 0.000,C 90.000,E1 3.784} C_DIS
LIN {X -0.037,Y -447.828,Z 1322.818,A 0.000,B 0.000,C 90.000,E1 3.212} C_DIS
LIN {X 0.136,Y -454.959,Z 1322.814,A 0.000,B 0.000,C 90.000,E1 2.465} C_DIS
LIN {X -0.079,Y -460.451,Z 1322.811,A 0.000,B 0.000,C 90.000,E1 1.892} C_DIS
LIN {X 0.116,Y -468.042,Z 1322.806,A 0.000,B 0.000,C 90.000,E1 0.974} C_DIS
LIN {X -0.227,Y -474.081,Z 1322.801,A 0.000,B 0.000,C 90.000,E1 0.229} C_DIS
LIN {X 0.112,Y -480.131,Z 1322.796,A 0.000,B 0.000,C 90.000,E1 359.312} C_DIS
LIN {X -0.126,Y -485.099,Z 1322.792,A 0.000,B 0.000,C 90.000,E1 358.568} C_DIS
LIN {X 0.184,Y -489.699,Z 1322.788,A 0.000,B 0.000,C 90.000,E1 357.764} C_DIS
LIN {X 0.028,Y -493.964,Z 1322.784,A 0.000,B 0.000,C 90.000,E1 357.020} C_DIS
LIN {X -0.241,Y -497.159,Z 1322.780,A 0.000,B 0.000,C 90.000,E1 356.445} C_DIS
LIN {X -0.121,Y -501.546,Z 1322.775,A 0.000,B 0.000,C 90.000,E1 355.527} C_DIS
LIN {X -0.143,Y -505.029,Z 1322.771,A 0.000,B 0.000,C 90.000,E1 354.780} C_DIS
LIN {X 0.174,Y -507.597,Z 1322.768,A 0.000,B 0.000,C 90.000,E1 354.147} C_DIS
LIN {X 0.261,Y -510.586,Z 1322.764,A 0.000,B 0.000,C 90.000,E1 353.394} C_DIS
LIN {X 0.111,Y -512.837,Z 1322.760,A 0.000,B 0.000,C 90.000,E1 352.818} C_DIS
LIN {X -0.053,Y -515.948,Z 1322.755,A 0.000,B 0.000,C 90.000,E1 351.951} C_DIS
LIN {X -0.188,Y -518.776,Z 1322.750,A 0.000,B 0.000,C 90.000,E1 351.084} C_DIS
LIN {X -0.208,Y -521.310,Z 1322.745,A 0.000,B 0.000,C 90.000,E1 350.208} C_DIS
LIN {X 0.222,Y -523.591,Z 1322.741,A 0.000,B 0.000,C 90.000,E1 349.285} C_DIS
LIN {X -0.258,Y -525.674,Z 1322.736,A 0.000,B 0.000,C 90.000,E1 348.465} C_DIS
LIN {X -0.065,Y -528.038,Z 1322.729,A 0.000,B 0.000,C 90.000,E1 347.285} C_DIS
LIN {X -0.010,Y -529.045,Z 1322.726,A 0.000,B 0.000,C 90.000,E1 346.700} C_DIS
LIN {X 0.241,Y -530.836,Z 1322.720,A 0.000,B 0.000,C 90.000,E1 345.519} C_DIS
LIN {X -0.032,Y -531.912,Z 1322.715,A 0.000,B 0.000,C 90.000,E1 344.685} C_DIS
LIN {X 0.038,Y -532.470,Z 1322.712,A 0.000,B 0.000,C 90.000,E1 344.102} C_DIS
LIN {X -0.034,Y -533.221,Z 1322.705,A 0.000,B 0.000,C 90.000,E1 342.960} C_DIS
LIN {X -0.287,Y -533.598,Z 1322.701,A 0.000,B 0.000,C 90.000,E1 342.127} C_DIS
LIN {X 0.105,Y -533.644,Z 1322.697,A 0.000,B 0.000,C 90.000,E1 341.511} C_DIS
LIN {X 0.047,Y -533.229,Z 1322.691,A 0.000,B 0.000,C 90.000,E1 340.369} C_DIS
LIN {X -0.042,Y -532.753,Z 1322.686,A 0.000,B 0.000,C 90.000,E1 339.518} C_DIS
LIN {X 0.056,Y -531.361,Z 1322.680,A 0.000,B 0.000,C 90.000,E1 338.358} C_DIS
LIN {X -0.052,Y -530.507,Z 1322.677,A 0.000,B 0.000,C 90.000,E1 337.794} C_DIS
LIN {X -0.094,Y -527.919,Z 1322.669,A 0.000,B 0.000,C 90.000,E1 336.357} C_DIS
LIN {X 0.085,Y -527.355,Z 1322.667,A 0.000,B 0.000,C 90.000,E1 336.049} C_DIS
LIN {X 0.122,Y -525.034,Z 1322.662,A 0.000,B 0.000,C 90.000,E1 335.177} C_DIS
LIN {X -0.282,Y -520.495,Z 1322.654,A 0.000,B 0.000,C 90.000,E1 333.768} C_DIS
LIN {X -0.094,Y -517.751,Z 1322.649,A 0.000,B 0.000,C 90.000,E1 332.871} C_DIS
LIN {X -0.028,Y -512.056,Z 1322.640,A 0.000,B 0.000,C 90.000,E1 331.101} C_DIS
LIN {X -0.051,Y -508.063,Z 1322.633,A 0.000,B 0.000,C 90.000,E1 329.921} C_DIS
LIN {X -0.087,Y -505.974,Z 1322.630,A 0.000,B 0.000,C 90.000,E1 329.331} C_DIS
LIN {X 0.052,Y -501.444,Z 1322.623,A 0.000,B 0.000,C 90.000,E1 328.122} C_DIS
LIN {X -0.168,Y -497.778,Z 1322.618,A 0.000,B 0.000,C 90.000,E1 327.248} C_DIS
LIN {X -0.230,Y -494.447,Z 1322.614,A 0.000,B 0.000,C 90.000,E1 326.501} C_DIS
LIN {X -0.112,Y -491.611,Z 1322.610,A 0.000,B 0.000,C 90.000,E1 325.881} C_DIS
LIN {X 0.203,Y -489.113,Z 1322.608,A 0.000,B 0.000,C 90.000,E1 325.388} C_DIS
LIN {X -0.016,Y -488.217,Z 1322.607,A 0.000,B 0.000,C 90.000,E1 325.261} C_DIS
LIN {X 0.045,Y -487.116,Z 1322.606,A 0.000,B 0.000,C 90.000,E1 325.102} C_DIS
LIN {X -0.178,Y -485.485,Z 1322.605,A 0.000,B 0.000,C 90.000,E1 324.975} C_DIS
LIN {X 0.043,Y -462.959,Z 1322.595,A 0.000,B 0.000,C 90.000,E1 323.004} C_DIS
LIN {X 0.193,Y -441.386,Z 1322.583,A 0.000,B 0.000,C 90.000,E1 320.884} C_DIS
LIN {X -0.064,Y -421.860,Z 1322.571,A 0.000,B 0.000,C 90.000,E1 318.771} C_DIS
LIN {X -0.010,Y -403.017,Z 1322.558,A 0.000,B 0.000,C 90.000,E1 316.419} C_DIS
LIN {X 0.028,Y -385.580,Z 1322.544,A 0.000,B 0.000,C 90.000,E1 313.947} C_DIS
LIN {X -0.153,Y -381.705,Z 1322.541,A 0.000,B 0.000,C 90.000,E1 313.380} C_DIS
LIN {X 0.088,Y -381.680,Z 1322.541,A 0.000,B 0.000,C 90.000,E1 313.338} C_DIS
LIN {X -0.119,Y -384.804,Z 1322.527,A 0.000,B 0.000,C 90.000,E1 310.906} C_DIS
LIN {X -0.130,Y -390.975,Z 1322.493,A 0.000,B 0.000,C 90.000,E1 304.818} C_DIS
LIN {X -0.062,Y -391.375,Z 1322.491,A 0.000,B 0.000,C 90.000,E1 304.452} C_DIS
LIN {X 0.206,Y -396.706,Z 1322.460,A 0.000,B 0.000,C 90.000,E1 298.743} C_DIS
LIN {X -0.114,Y -397.080,Z 1322.458,A 0.000,B 0.000,C 90.000,E1 298.437} C_DIS
LIN {X -0.159,Y -401.504,Z 1322.427,A 0.000,B 0.000,C 90.000,E1 292.823} C_DIS
LIN {X 0.159,Y -401.771,Z 1322.423,A 0.000,B 0.000,C 90.000,E1 292.078} C_DIS
LIN {X -0.033,Y -404.578,Z 1322.396,A 0.000,B 0.000,C 90.000,E1 287.221} C_DIS
LIN {X 0.068,Y -404.759,Z 1322.394,A 0.000,B 0.000,C 90.000,E1 286.858} C_DIS
LIN {X -0.025,Y -406.047,Z 1322.365,A 0.000,B 0.000,C 90.000,E1 281.658} C_DIS
LIN {X 0.064,Y -406.132,Z 1322.363,A 0.000,B 0.000,C 90.000,E1 281.299} C_DIS
LIN {X 0.095,Y -405.658,Z 1322.334,A 0.000,B 0.000,C 90.000,E1 276.087} C_DIS
LIN {X 0.100,Y -405.591,Z 1322.332,A 0.000,B 0.000,C 90.000,E1 275.739} C_DIS
LIN {X 0.174,Y -403.545,Z 1322.305,A 0.000,B 0.000,C 90.000,E1 270.859} C_DIS
LIN {X 0.108,Y -403.024,Z 1322.301,A 0.000,B 0.000,C 90.000,E1 270.172} C_DIS
LIN {X -0.070,Y -399.002,Z 1322.272,A 0.000,B 0.000,C 90.000,E1 264.951} C_DIS
LIN {X 0.092,Y -392.912,Z 1322.241,A 0.000,B 0.000,C 90.000,E1 259.285} C_DIS
LIN {X 0.082,Y -391.846,Z 1322.237,A 0.000,B 0.000,C 90.000,E1 258.578} C_DIS
LIN {X -0.162,Y -385.717,Z 1322.211,A 0.000,B 0.000,C 90.000,E1 253.976} C_DIS
LIN {X -0.115,Y -384.941,Z 1322.207,A 0.000,B 0.000,C 90.000,E1 253.251} C_DIS
LIN {X 0.001,Y -378.094,Z 1322.183,A 0.000,B 0.000,C 90.000,E1 248.901} C_DIS
LIN {X 0.085,Y -376.338,Z 1322.175,A 0.000,B 0.000,C 90.000,E1 247.433} C_DIS
LIN {X -0.137,Y -375.824,Z 1322.173,A 0.000,B 0.000,C 90.000,E1 247.102} C_DIS
LIN {X -0.019,Y -369.062,Z 1322.150,A 0.000,B 0.000,C 90.000,E1 243.050} C_DIS
LIN {X -0.107,Y -366.213,Z 1322.138,A 0.000,B 0.000,C 90.000,E1 240.845} C_DIS
LIN {X 0.055,Y -358.809,Z 1322.113,A 0.000,B 0.000,C 90.000,E1 236.342} C_DIS
LIN {X 0.133,Y -356.001,Z 1322.101,A 0.000,B 0.000,C 90.000,E1 234.069} C_DIS
LIN {X -0.037,Y -352.666,Z 1322.090,A 0.000,B 0.000,C 90.000,E1 232.145} C_DIS
LIN {X 0.161,Y -352.663,Z 1322.090,A 0.000,B 0.000,C 90.000,E1 232.110} C_DIS
LIN {X 0.114,Y -366.235,Z 1322.075,A 0.000,B 0.000,C 90.000,E1 229.542} C_DIS
LIN {X -0.005,Y -381.666,Z 1322.061,A 0.000,B 0.000,C 90.000,E1 226.986} C_DIS
LIN {X -0.229,Y -398.763,Z 1322.047,A 0.000,B 0.000,C 90.000,E1 224.514} C_DIS
LIN {X -0.152,Y -417.577,Z 1322.034,A 0.000,B 0.000,C 90.000,E1 222.081} C_DIS
LIN {X 0.138,Y -437.303,Z 1322.021,A 0.000,B 0.000,C 90.000,E1 219.806} C_DIS
LIN {X 0.186,Y -442.977,Z 1322.018,A 0.000,B 0.000,C 90.000,E1 219.197} C_DIS
LIN {X 0.014,Y -444.627,Z 1322.016,A 0.000,B 0.000,C 90.000,E1 218.910} C_DIS
LIN {X -0.024,Y -445.787,Z 1322.014,A 0.000,B 0.000,C 90.000,E1 218.588} C_DIS
LIN {X 0.015,Y -446.692,Z 1322.013,A 0.000,B 0.000,C 90.000,E1 218.257} C_DIS
LIN {X 0.035,Y -448.065,Z 1322.009,A 0.000,B 0.000,C 90.000,E1 217.604} C_DIS
LIN {X 0.065,Y -449.136,Z 1322.005,A 0.000,B 0.000,C 90.000,E1 216.950} C_DIS
LIN {X 0.104,Y -449.951,Z 1322.002,A 0.000,B 0.000,C 90.000,E1 216.297} C_DIS
LIN {X 0.221,Y -450.847,Z 1321.996,A 0.000,B 0.000,C 90.000,E1 215.311} C_DIS
LIN {X 0.034,Y -453.338,Z 1321.982,A 0.000,B 0.000,C 90.000,E1 212.752} C_DIS
LIN {X 0.238,Y -455.492,Z 1321.971,A 0.000,B 0.000,C 90.000,E1 210.797} C_DIS
LIN {X 0.145,Y -458.195,Z 1321.959,A 0.000,B 0.000,C 90.000,E1 208.565} C_DIS
LIN {X -0.061,Y -462.171,Z 1321.943,A 0.000,B 0.000,C 90.000,E1 205.720} C_DIS
LIN {X -0.189,Y -465.407,Z 1321.931,A 0.000,B 0.000,C 90.000,E1 203.515} C_DIS
LIN {X 0.118,Y -467.608,Z 1321.922,A 0.000,B 0.000,C 90.000,E1 201.897} C_DIS
LIN {X -0.096,Y -469.182,Z 1321.915,A 0.000,B 0.000,C 90.000,E1 200.663} C_DIS
LIN {X -0.098,Y -471.739,Z 1321.904,A 0.000,B 0.000,C 90.000,E1 198.779} C_DIS
LIN {X -0.152,Y -473.870,Z 1321.896,A 0.000,B 0.000,C 90.000,E1 197.221} C_DIS
LIN {X 0.127,Y -476.287,Z 1321.885,A 0.000,B 0.000,C 90.000,E1 195.315} C_DIS
LIN {X -0.161,Y -479.083,Z 1321.873,A 0.000,B 0.000,C 90.000,E1 193.175} C_DIS
LIN {X -0.145,Y -481.819,Z 1321.861,A 0.000,B 0.000,C 90.000,E1 191.007} C_DIS
LIN {X 0.250,Y -483.360,Z 1321.854,A 0.000,B 0.000,C 90.000,E1 189.726} C_DIS
LIN {X -0.217,Y -485.657,Z 1321.844,A 0.000,B 0.000,C 90.000,E1 187.936} C_DIS
LIN {X 0.039,Y -487.429,Z 1321.835,A 0.000,B 0.000,C 90.000,E1 186.372} C_DIS
LIN {X 0.222,Y -489.001,Z 1321.827,A 0.000,B 0.000,C 90.000,E1 184.821} C_DIS
LIN {X 0.115,Y -490.096,Z 1321.820,A 0.000,B 0.000,C 90.000,E1 183.612} C_DIS
LIN {X -0.011,Y -491.010,Z 1321.813,A 0.000,B 0.000,C 90.000,E1 182.407} C_DIS
LIN {X -0.125,Y -491.789,Z 1321.807,A 0.000,B 0.000,C 90.000,E1 181.203} C_DIS
LIN {X 0.061,Y -492.100,Z 1321.803,A 0.000,B 0.000,C 90.000,E1 180.573} C_DIS
LIN {X -0.198,Y -492.606,Z 1321.795,A 0.000,B 0.000,C 90.000,E1 179.083} C_DIS
LIN {X -0.142,Y -492.641,Z 1321.790,A 0.000,B 0.000,C 90.000,E1 178.165} C_DIS
LIN {X -0.100,Y -492.563,Z 1321.785,A 0.000,B 0.000,C 90.000,E1 177.249} C_DIS
LIN {X -0.039,Y -492.342,Z 1321.780,A 0.000,B 0.000,C 90.000,E1 176.331} C_DIS
LIN {X 0.018,Y -491.828,Z 1321.775,A 0.000,B 0.000,C 90.000,E1 175.412} C_DIS
LIN {X 0.113,Y -491.152,Z 1321.770,A 0.000,B 0.000,C 90.000,E1 174.489} C_DIS
LIN {X 0.035,Y -489.937,Z 1321.763,A 0.000,B 0.000,C 90.000,E1 173.280} C_DIS
LIN {X 0.113,Y -488.649,Z 1321.758,A 0.000,B 0.000,C 90.000,E1 172.356} C_DIS
LIN {X 0.173,Y -487.155,Z 1321.753,A 0.000,B 0.000,C 90.000,E1 171.432} C_DIS
LIN {X -0.068,Y -485.999,Z 1321.749,A 0.000,B 0.000,C 90.000,E1 170.849} C_DIS
LIN {X -0.173,Y -483.140,Z 1321.742,A 0.000,B 0.000,C 90.000,E1 169.634} C_DIS
LIN {X 0.036,Y -481.430,Z 1321.739,A 0.000,B 0.000,C 90.000,E1 168.993} C_DIS
LIN {X 0.183,Y -478.233,Z 1321.734,A 0.000,B 0.000,C 90.000,E1 168.049} C_DIS
LIN {X 0.037,Y -477.081,Z 1321.732,A 0.000,B 0.000,C 90.000,E1 167.757} C_DIS
LIN {X 0.030,Y -472.628,Z 1321.727,A 0.000,B 0.000,C 90.000,E1 166.825} C_DIS
LIN {X 0.057,Y -469.820,Z 1321.724,A 0.000,B 0.000,C 90.000,E1 166.353} C_DIS
LIN {X -0.016,Y -462.050,Z 1321.717,A 0.000,B 0.000,C 90.000,E1 165.102} C_DIS
LIN {X -0.157,Y -453.469,Z 1321.709,A 0.000,B 0.000,C 90.000,E1 163.685} C_DIS
LIN {X 0.067,Y -448.694,Z 1321.705,A 0.000,B 0.000,C 90.000,E1 162.851} C_DIS
LIN {X -0.046,Y -444.506,Z 1321.700,A 0.000,B 0.000,C 90.000,E1 162.054} C_DIS
LIN {X 0.087,Y -441.269,Z 1321.696,A 0.000,B 0.000,C 90.000,E1 161.221} C_DIS
LIN {X -0.195,Y -440.852,Z 1321.695,A 0.000,B 0.000,C 90.000,E1 161.094} C_DIS
LIN {X 0.073,Y -439.900,Z 1321.692,A 0.000,B 0.000,C 90.000,E1 160.496} C_DIS
LIN {X -0.212,Y -439.790,Z 1321.691,A 0.000,B 0.000,C 90.000,E1 160.369} C_DIS
LIN {X 0.105,Y -440.015,Z 1321.689,A 0.000,B 0.000,C 90.000,E1 160.061} C_DIS
LIN {X 0.027,Y -440.035,Z 1321.689,A 0.000,B 0.000,C 90.000,E1 160.061} C_DIS
LIN {X -0.013,Y -440.067,Z 1321.689,A 0.000,B 0.000,C 90.000,E1 160.061} C_DIS
LIN {X -0.239,Y -441.510,Z 1321.688,A 0.000,B 0.000,C 90.000,E1 159.880} C_DIS
LIN {X 0.107,Y -442.506,Z 1321.687,A 0.000,B 0.000,C 90.000,E1 159.645} C_DIS
LIN {X 0.067,Y -442.557,Z 1321.687,A 0.000,B 0.000,C 90.000,E1 159.645} C_DIS
LIN {X 0.001,Y -445.559,Z 1321.686,A 0.000,B 0.000,C 90.000,E1 159.390} C_DIS
LIN {X 0.131,Y -450.146,Z 1321.683,A 0.000,B 0.000,C 90.000,E1 158.954} C_DIS
LIN {X -0.084,Y -460.517,Z 1321.679,A 0.000,B 0.000,C 90.000,E1 158.156} C_DIS
LIN {X 0.103,Y -472.820,Z 1321.673,A 0.000,B 0.000,C 90.000,E1 157.177} C_DIS
LIN {X 0.003,Y -481.550,Z 1321.669,A 0.000,B 0.000,C 90.000,E1 156.485} C_DIS
LIN {X 0.130,Y -487.457,Z 1321.667,A 0.000,B 0.000,C 90.000,E1 155.973} C_DIS
LIN {X -0.186,Y -494.563,Z 1321.663,A 0.000,B 0.000,C 90.000,E1 155.357} C_DIS
LIN {X -0.055,Y -501.494,Z 1321.659,A 0.000,B 0.000,C 90.000,E1 154.665} C_DIS
LIN {X 0.032,Y -506.877,Z 1321.656,A 0.000,B 0.000,C 90.000,E1 154.101} C_DIS
LIN {X 0.062,Y -513.273,Z 1321.652,A 0.000,B 0.000,C 90.000,E1 153.384} C_DIS
LIN {X 0.040,Y -517.018,Z 1321.650,A 0.000,B 0.000,C 90.000,E1 152.948} C_DIS
LIN {X 0.235,Y -520.548,Z 1321.647,A 0.000,B 0.000,C 90.000,E1 152.487} C_DIS
LIN {X 0.289,Y -524.691,Z 1321.644,A 0.000,B 0.000,C 90.000,E1 151.897} C_DIS
LIN {X -0.342,Y -528.363,Z 1321.641,A 0.000,B 0.000,C 90.000,E1 151.385} C_DIS
LIN {X 0.341,Y -532.091,Z 1321.637,A 0.000,B 0.000,C 90.000,E1 150.589} C_DIS
LIN {X -0.102,Y -533.911,Z 1321.635,A 0.000,B 0.000,C 90.000,E1 150.205} C_DIS
LIN {X -0.127,Y -535.021,Z 1321.633,A 0.000,B 0.000,C 90.000,E1 149.921} C_DIS
LIN {X 0.031,Y -536.979,Z 1321.630,A 0.000,B 0.000,C 90.000,E1 149.331} C_DIS
LIN {X 0.200,Y -539.364,Z 1321.625,A 0.000,B 0.000,C 90.000,E1 148.456} C_DIS
LIN {X -0.350,Y -541.322,Z 1321.620,A 0.000,B 0.000,C 90.000,E1 147.661} C_DIS
LIN {X 0.159,Y -542.888,Z 1321.615,A 0.000,B 0.000,C 90.000,E1 146.755} C_DIS
LIN {X -0.061,Y -544.171,Z 1321.611,A 0.000,B 0.000,C 90.000,E1 145.928} C_DIS
LIN {X 0.212,Y -545.519,Z 1321.604,A 0.000,B 0.000,C 90.000,E1 144.769} C_DIS
LIN {X 0.047,Y -546.636,Z 1321.598,A 0.000,B 0.000,C 90.000,E1 143.657} C_DIS
LIN {X -0.125,Y -548.069,Z 1321.589,A 0.000,B 0.000,C 90.000,E1 141.984} C_DIS
LIN {X -0.032,Y -548.638,Z 1321.586,A 0.000,B 0.000,C 90.000,E1 141.412} C_DIS
LIN {X -0.016,Y -549.772,Z 1321.583,A 0.000,B 0.000,C 90.000,E1 140.848} C_DIS
LIN {X -0.005,Y -550.208,Z 1321.582,A 0.000,B 0.000,C 90.000,E1 140.723} C_DIS
LIN {X 0.055,Y -551.354,Z 1321.581,A 0.000,B 0.000,C 90.000,E1 140.642} C_DIS
LIN {X -0.071,Y -557.009,Z 1321.580,A 0.000,B 0.000,C 90.000,E1 140.436} C_DIS
LIN {X -0.075,Y -567.268,Z 1321.578,A 0.000,B 0.000,C 90.000,E1 140.114} C_DIS
LIN {X 0.015,Y -570.619,Z 1321.578,A 0.000,B 0.000,C 90.000,E1 139.989} C_DIS
LIN {X 0.015,Y -576.355,Z 1321.576,A 0.000,B 0.000,C 90.000,E1 139.703} C_DIS
LIN {X -0.226,Y -582.297,Z 1321.574,A 0.000,B 0.000,C 90.000,E1 139.380} C_DIS
LIN {X -0.260,Y -590.755,Z 1321.571,A 0.000,B 0.000,C 90.000,E1 138.771} C_DIS
LIN {X -0.003,Y -593.497,Z 1321.570,A 0.000,B 0.000,C 90.000,E1 138.528} C_DIS
LIN {X 0.142,Y -597.422,Z 1321.568,A 0.000,B 0.000,C 90.000,E1 138.162} C_DIS
LIN {X -0.033,Y -603.602,Z 1321.564,A 0.000,B 0.000,C 90.000,E1 137.553} C_DIS
LIN {X -0.200,Y -606.149,Z 1321.563,A 0.000,B 0.000,C 90.000,E1 137.310} C_DIS
LIN {X 0.263,Y -611.631,Z 1321.559,A 0.000,B 0.000,C 90.000,E1 136.620} C_DIS
LIN {X -0.088,Y -615.773,Z 1321.556,A 0.000,B 0.000,C 90.000,E1 136.134} C_DIS
LIN {X 0.101,Y -618.657,Z 1321.554,A 0.000,B 0.000,C 90.000,E1 135.729} C_DIS
LIN {X 0.294,Y -624.896,Z 1321.549,A 0.000,B 0.000,C 90.000,E1 134.838} C_DIS
LIN {X 0.007,Y -629.208,Z 1321.546,A 0.000,B 0.000,C 90.000,E1 134.231} C_DIS
LIN {X -0.028,Y -638.033,Z 1321.538,A 0.000,B 0.000,C 90.000,E1 132.852} C_DIS
LIN {X -0.211,Y -646.144,Z 1321.531,A 0.000,B 0.000,C 90.000,E1 131.515} C_DIS
LIN {X 0.066,Y -650.618,Z 1321.526,A 0.000,B 0.000,C 90.000,E1 130.744} C_DIS
LIN {X -0.086,Y -656.251,Z 1321.521,A 0.000,B 0.000,C 90.000,E1 129.769} C_DIS
LIN {X 0.345,Y -661.591,Z 1321.516,A 0.000,B 0.000,C 90.000,E1 128.749} C_DIS
LIN {X -0.082,Y -666.484,Z 1321.510,A 0.000,B 0.000,C 90.000,E1 127.810} C_DIS
LIN {X -0.009,Y -668.721,Z 1321.507,A 0.000,B 0.000,C 90.000,E1 127.317} C_DIS
LIN {X 0.083,Y -670.917,Z 1321.505,A 0.000,B 0.000,C 90.000,E1 126.824} C_DIS
LIN {X -0.233,Y -674.793,Z 1321.499,A 0.000,B 0.000,C 90.000,E1 125.884} C_DIS
LIN {X 0.044,Y -678.243,Z 1321.494,A 0.000,B 0.000,C 90.000,E1 124.898} C_DIS
LIN {X -0.193,Y -680.518,Z 1321.490,A 0.000,B 0.000,C 90.000,E1 124.199} C_DIS
LIN {X 0.149,Y -683.109,Z 1321.485,A 0.000,B 0.000,C 90.000,E1 123.214} C_DIS
LIN {X 0.155,Y -684.865,Z 1321.481,A 0.000,B 0.000,C 90.000,E1 122.498} C_DIS
LIN {X -0.030,Y -686.426,Z 1321.477,A 0.000,B 0.000,C 90.000,E1 121.799} C_DIS
LIN {X 0.005,Y -688.206,Z 1321.471,A 0.000,B 0.000,C 90.000,E1 120.846} C_DIS
LIN {X 0.077,Y -689.320,Z 1321.467,A 0.000,B 0.000,C 90.000,E1 120.129} C_DIS
LIN {X -0.205,Y -690.558,Z 1321.462,A 0.000,B 0.000,C 90.000,E1 119.205} C_DIS
LIN {X -0.239,Y -691.324,Z 1321.456,A 0.000,B 0.000,C 90.000,E1 118.025} C_DIS
LIN {X 0.105,Y -691.585,Z 1321.450,A 0.000,B 0.000,C 90.000,E1 117.052} C_DIS
LIN {X -0.101,Y -691.630,Z 1321.446,A 0.000,B 0.000,C 90.000,E1 116.360} C_DIS
LIN {X -0.001,Y -691.314,Z 1321.443,A 0.000,B 0.000,C 90.000,E1 115.643} C_DIS
LIN {X 0.181,Y -690.982,Z 1321.440,A 0.000,B 0.000,C 90.000,E1 115.155} C_DIS
LIN {X 0.031,Y -690.340,Z 1321.437,A 0.000,B 0.000,C 90.000,E1 114.695} C_DIS
LIN {X -0.021,Y -689.924,Z 1321.436,A 0.000,B 0.000,C 90.000,E1 114.463} C_DIS
LIN {X -0.182,Y -688.616,Z 1321.433,A 0.000,B 0.000,C 90.000,E1 114.003} C_DIS
LIN {X -0.231,Y -687.568,Z 1321.432,A 0.000,B 0.000,C 90.000,E1 113.770} C_DIS
LIN {X 0.106,Y -685.763,Z 1321.430,A 0.000,B 0.000,C 90.000,E1 113.387} C_DIS
LIN {X 0.217,Y -685.038,Z 1321.429,A 0.000,B 0.000,C 90.000,E1 113.259} C_DIS
LIN {X 0.054,Y -683.943,Z 1321.429,A 0.000,B 0.000,C 90.000,E1 113.153} C_DIS
LIN {X 0.045,Y -678.877,Z 1321.426,A 0.000,B 0.000,C 90.000,E1 112.695} C_DIS
LIN {X -0.053,Y -676.830,Z 1321.426,A 0.000,B 0.000,C 90.000,E1 112.589} C_DIS
LIN {X 0.054,Y -672.422,Z 1321.425,A 0.000,B 0.000,C 90.000,E1 112.408} C_DIS
LIN {X 0.089,Y -669.173,Z 1321.424,A 0.000,B 0.000,C 90.000,E1 112.280} C_DIS
LIN {X -0.251,Y -666.013,Z 1321.423,A 0.000,B 0.000,C 90.000,E1 112.206} C_DIS
LIN {X 0.244,Y -661.233,Z 1321.423,A 0.000,B 0.000,C 90.000,E1 112.078} C_DIS
LIN {X -0.101,Y -656.030,Z 1321.422,A 0.000,B 0.000,C 90.000,E1 112.025} C_DIS
LIN {X 0.302,Y -646.711,Z 1321.422,A 0.000,B 0.000,C 90.000,E1 111.897} C_DIS
LIN {X -0.191,Y -643.657,Z 1321.422,A 0.000,B 0.000,C 90.000,E1 111.897} C_DIS
LIN {X -0.149,Y -642.120,Z 1321.421,A 0.000,B 0.000,C 90.000,E1 111.844} C_DIS
LIN {X -0.188,Y -642.117,Z 1321.421,A 0.000,B 0.000,C 90.000,E1 111.844} C_DIS
LIN {X 0.336,Y -643.251,Z 1321.420,A 0.000,B 0.000,C 90.000,E1 111.589} C_DIS
LIN {X 0.261,Y -648.336,Z 1321.417,A 0.000,B 0.000,C 90.000,E1 110.972} C_DIS
LIN {X 0.144,Y -651.253,Z 1321.415,A 0.000,B 0.000,C 90.000,E1 110.610} C_DIS
LIN {X -0.049,Y -656.228,Z 1321.411,A 0.000,B 0.000,C 90.000,E1 109.885} C_DIS
LIN {X -0.025,Y -659.872,Z 1321.407,A 0.000,B 0.000,C 90.000,E1 109.268} C_DIS
LIN {X -0.135,Y -663.485,Z 1321.403,A 0.000,B 0.000,C 90.000,E1 108.544} C_DIS
LIN {X -0.216,Y -666.587,Z 1321.399,A 0.000,B 0.000,C 90.000,E1 107.819} C_DIS
LIN {X -0.188,Y -668.470,Z 1321.396,A 0.000,B 0.000,C 90.000,E1 107.330} C_DIS
LIN {X 0.222,Y -670.972,Z 1321.392,A 0.000,B 0.000,C 90.000,E1 106.567} C_DIS
LIN {X 0.276,Y -672.496,Z 1321.390,A 0.000,B 0.000,C 90.000,E1 106.079} C_DIS
LIN {X 0.092,Y -674.380,Z 1321.385,A 0.000,B 0.000,C 90.000,E1 105.371} C_DIS
LIN {X -0.071,Y -675.926,Z 1321.381,A 0.000,B 0.000,C 90.000,E1 104.662} C_DIS
LIN {X -0.052,Y -677.258,Z 1321.377,A 0.000,B 0.000,C 90.000,E1 103.939} C_DIS
LIN {X -0.147,Y -677.898,Z 1321.375,A 0.000,B 0.000,C 90.000,E1 103.467} C_DIS
LIN {X -0.390,Y -678.360,Z 1321.372,A 0.000,B 0.000,C 90.000,E1 103.008} C_DIS
LIN {X 0.145,Y -678.712,Z 1321.368,A 0.000,B 0.000,C 90.000,E1 102.243} C_DIS
LIN {X 0.061,Y -678.780,Z 1321.365,A 0.000,B 0.000,C 90.000,E1 101.771} C_DIS
LIN {X -0.027,Y -678.617,Z 1321.363,A 0.000,B 0.000,C 90.000,E1 101.299} C_DIS
LIN {X -0.247,Y -678.256,Z 1321.360,A 0.000,B 0.000,C 90.000,E1 100.838} C_DIS
LIN {X 0.326,Y -677.682,Z 1321.357,A 0.000,B 0.000,C 90.000,E1 100.310} C_DIS
LIN {X 0.108,Y -676.910,Z 1321.355,A 0.000,B 0.000,C 90.000,E1 99.849} C_DIS
LIN {X -0.168,Y -675.163,Z 1321.351,A 0.000,B 0.000,C 90.000,E1 99.151} C_DIS
LIN {X -0.291,Y -673.627,Z 1321.348,A 0.000,B 0.000,C 90.000,E1 98.681} C_DIS
LIN {X 0.136,Y -671.744,Z 1321.345,A 0.000,B 0.000,C 90.000,E1 98.163} C_DIS
LIN {X -0.110,Y -669.633,Z 1321.343,A 0.000,B 0.000,C 90.000,E1 97.701} C_DIS
LIN {X 0.201,Y -666.073,Z 1321.339,A 0.000,B 0.000,C 90.000,E1 96.947} C_DIS
LIN {X -0.084,Y -663.484,Z 1321.336,A 0.000,B 0.000,C 90.000,E1 96.486} C_DIS
LIN {X 0.176,Y -659.921,Z 1321.333,A 0.000,B 0.000,C 90.000,E1 95.853} C_DIS
LIN {X -0.147,Y -656.838,Z 1321.330,A 0.000,B 0.000,C 90.000,E1 95.391} C_DIS
LIN {X 0.104,Y -653.529,Z 1321.327,A 0.000,B 0.000,C 90.000,E1 94.878} C_DIS
LIN {X 0.284,Y -648.897,Z 1321.324,A 0.000,B 0.000,C 90.000,E1 94.245} C_DIS
LIN {X -0.109,Y -645.009,Z 1321.321,A 0.000,B 0.000,C 90.000,E1 93.784} C_DIS
LIN {X -0.044,Y -639.622,Z 1321.318,A 0.000,B 0.000,C 90.000,E1 93.154} C_DIS
LIN {X 0.137,Y -635.057,Z 1321.315,A 0.000,B 0.000,C 90.000,E1 92.636} C_DIS
LIN {X 0.287,Y -630.184,Z 1321.312,A 0.000,B 0.000,C 90.000,E1 92.121} C_DIS
LIN {X -0.170,Y -623.878,Z 1321.309,A 0.000,B 0.000,C 90.000,E1 91.547} C_DIS
LIN {X 0.178,Y -617.316,Z 1321.305,A 0.000,B 0.000,C 90.000,E1 90.917} C_DIS
LIN {X 0.127,Y -615.926,Z 1321.305,A 0.000,B 0.000,C 90.000,E1 90.802} C_DIS
LIN {X 0.015,Y -608.886,Z 1321.302,A 0.000,B 0.000,C 90.000,E1 90.286} C_DIS
LIN {X 0.143,Y -602.384,Z 1321.299,A 0.000,B 0.000,C 90.000,E1 89.885} C_DIS
LIN {X 0.142,Y -595.768,Z 1321.298,A 0.000,B 0.000,C 90.000,E1 89.542} C_DIS
LIN {X -0.039,Y -588.788,Z 1321.296,A 0.000,B 0.000,C 90.000,E1 89.255} C_DIS
LIN {X -0.143,Y -576.830,Z 1321.293,A 0.000,B 0.000,C 90.000,E1 88.797} C_DIS
LIN {X 0.019,Y -574.955,Z 1321.293,A 0.000,B 0.000,C 90.000,E1 88.682} C_DIS
LIN {X 0.276,Y -572.971,Z 1321.292,A 0.000,B 0.000,C 90.000,E1 88.511} C_DIS
LIN {X -0.101,Y -572.170,Z 1321.291,A 0.000,B 0.000,C 90.000,E1 88.453} C_DIS
LIN {X -0.143,Y -572.159,Z 1321.291,A 0.000,B 0.000,C 90.000,E1 88.453} C_DIS
LIN {X 0.250,Y -571.575,Z 1321.290,A 0.000,B 0.000,C 90.000,E1 88.167} C_DIS
LIN {X 0.051,Y -571.435,Z 1321.289,A 0.000,B 0.000,C 90.000,E1 88.051} C_DIS
LIN {X -0.032,Y -571.473,Z 1321.287,A 0.000,B 0.000,C 90.000,E1 87.650} C_DIS
LIN {X -0.039,Y -573.478,Z 1321.275,A 0.000,B 0.000,C 90.000,E1 85.469} C_DIS
LIN {X 0.103,Y -575.868,Z 1321.263,A 0.000,B 0.000,C 90.000,E1 83.280} C_DIS
LIN {X 0.044,Y -577.863,Z 1321.254,A 0.000,B 0.000,C 90.000,E1 81.659} C_DIS
LIN {X 0.023,Y -579.730,Z 1321.245,A 0.000,B 0.000,C 90.000,E1 80.038} C_DIS
LIN {X -0.216,Y -580.967,Z 1321.239,A 0.000,B 0.000,C 90.000,E1 78.982} C_DIS
LIN {X 0.018,Y -582.065,Z 1321.233,A 0.000,B 0.000,C 90.000,E1 77.881} C_DIS
LIN {X -0.188,Y -583.063,Z 1321.227,A 0.000,B 0.000,C 90.000,E1 76.825} C_DIS
LIN {X 0.227,Y -584.283,Z 1321.218,A 0.000,B 0.000,C 90.000,E1 75.172} C_DIS
LIN {X 0.261,Y -585.396,Z 1321.209,A 0.000,B 0.000,C 90.000,E1 73.559} C_DIS
LIN {X 0.089,Y -586.279,Z 1321.201,A 0.000,B 0.000,C 90.000,E1 72.236} C_DIS
LIN {X 0.349,Y -587.358,Z 1321.193,A 0.000,B 0.000,C 90.000,E1 70.604} C_DIS
LIN {X 0.030,Y -588.858,Z 1321.179,A 0.000,B 0.000,C 90.000,E1 68.230} C_DIS
LIN {X 0.200,Y -589.894,Z 1321.170,A 0.000,B 0.000,C 90.000,E1 66.613} C_DIS
LIN {X -0.151,Y -591.018,Z 1321.161,A 0.000,B 0.000,C 90.000,E1 65.049} C_DIS
LIN {X -0.066,Y -592.356,Z 1321.151,A 0.000,B 0.000,C 90.000,E1 63.179} C_DIS
LIN {X 0.158,Y -593.647,Z 1321.142,A 0.000,B 0.000,C 90.000,E1 61.563} C_DIS
LIN {X -0.215,Y -595.366,Z 1321.132,A 0.000,B 0.000,C 90.000,E1 59.744} C_DIS
LIN {X 0.139,Y -596.971,Z 1321.123,A 0.000,B 0.000,C 90.000,E1 58.122} C_DIS
LIN {X -0.067,Y -598.946,Z 1321.113,A 0.000,B 0.000,C 90.000,E1 56.294} C_DIS
LIN {X 0.195,Y -600.588,Z 1321.104,A 0.000,B 0.000,C 90.000,E1 54.689} C_DIS
LIN {X -0.248,Y -601.809,Z 1321.097,A 0.000,B 0.000,C 90.000,E1 53.417} C_DIS
LIN {X 0.166,Y -602.974,Z 1321.089,A 0.000,B 0.000,C 90.000,E1 52.065} C_DIS
LIN {X 0.241,Y -603.755,Z 1321.084,A 0.000,B 0.000,C 90.000,E1 51.009} C_DIS
LIN {X -0.001,Y -604.817,Z 1321.075,A 0.000,B 0.000,C 90.000,E1 49.461} C_DIS
LIN {X 0.105,Y -605.256,Z 1321.069,A 0.000,B 0.000,C 90.000,E1 48.405} C_DIS
LIN {X -0.236,Y -605.444,Z 1321.063,A 0.000,B 0.000,C 90.000,E1 47.391} C_DIS
LIN {X -0.105,Y -605.654,Z 1321.054,A 0.000,B 0.000,C 90.000,E1 45.810} C_DIS
LIN {X 0.174,Y -605.655,Z 1321.050,A 0.000,B 0.000,C 90.000,E1 45.000} C_DIS
LIN {X 0.259,Y -605.401,Z 1321.044,A 0.000,B 0.000,C 90.000,E1 43.947} C_DIS
LIN {X 0.116,Y -605.198,Z 1321.040,A 0.000,B 0.000,C 90.000,E1 43.176} C_DIS
LIN {X -0.015,Y -604.808,Z 1321.033,A 0.000,B 0.000,C 90.000,E1 41.881} C_DIS
LIN {X 0.340,Y -604.319,Z 1321.025,A 0.000,B 0.000,C 90.000,E1 40.539} C_DIS
LIN {X 0.098,Y -603.547,Z 1321.017,A 0.000,B 0.000,C 90.000,E1 38.991} C_DIS
LIN {X -0.076,Y -603.147,Z 1321.012,A 0.000,B 0.000,C 90.000,E1 38.222} C_DIS
LIN {X -0.157,Y -602.590,Z 1321.008,A 0.000,B 0.000,C 90.000,E1 37.443} C_DIS
LIN {X -0.238,Y -601.779,Z 1321.004,A 0.000,B 0.000,C 90.000,E1 36.664} C_DIS
LIN {X 0.028,Y -600.742,Z 1320.999,A 0.000,B 0.000,C 90.000,E1 35.851} C_DIS
LIN {X -0.178,Y -599.115,Z 1320.993,A 0.000,B 0.000,C 90.000,E1 34.818} C_DIS
LIN {X -0.399,Y -597.224,Z 1320.988,A 0.000,B 0.000,C 90.000,E1 33.785} C_DIS
LIN {X -0.042,Y -595.585,Z 1320.983,A 0.000,B 0.000,C 90.000,E1 32.959} C_DIS
LIN {X 0.188,Y -592.978,Z 1320.977,A 0.000,B 0.000,C 90.000,E1 31.878} C_DIS
LIN {X -0.322,Y -590.694,Z 1320.973,A 0.000,B 0.000,C 90.000,E1 31.131} C_DIS
LIN {X -0.350,Y -588.064,Z 1320.968,A 0.000,B 0.000,C 90.000,E1 30.335} C_DIS
LIN {X 0.107,Y -585.044,Z 1320.964,A 0.000,B 0.000,C 90.000,E1 29.489} C_DIS
LIN {X 0.021,Y -581.634,Z 1320.959,A 0.000,B 0.000,C 90.000,E1 28.693} C_DIS
LIN {X -0.037,Y -578.480,Z 1320.956,A 0.000,B 0.000,C 90.000,E1 28.025} C_DIS
LIN {X 0.113,Y -575.009,Z 1320.952,A 0.000,B 0.000,C 90.000,E1 27.334} C_DIS
LIN {X -0.016,Y -571.212,Z 1320.948,A 0.000,B 0.000,C 90.000,E1 26.668} C_DIS
LIN {X 0.075,Y -567.139,Z 1320.944,A 0.000,B 0.000,C 90.000,E1 25.976} C_DIS
LIN {X 0.131,Y -562.730,Z 1320.941,A 0.000,B 0.000,C 90.000,E1 25.283} C_DIS
LIN {X -0.208,Y -558.967,Z 1320.938,A 0.000,B 0.000,C 90.000,E1 24.771} C_DIS
LIN {X -0.134,Y -553.852,Z 1320.934,A 0.000,B 0.000,C 90.000,E1 24.079} C_DIS
LIN {X 0.019,Y -549.585,Z 1320.931,A 0.000,B 0.000,C 90.000,E1 23.515} C_DIS
LIN {X 0.044,Y -544.930,Z 1320.928,A 0.000,B 0.000,C 90.000,E1 22.950} C_DIS
LIN {X -0.021,Y -536.457,Z 1320.922,A 0.000,B 0.000,C 90.000,E1 21.972} C_DIS
LIN {X -0.045,Y -531.274,Z 1320.919,A 0.000,B 0.000,C 90.000,E1 21.408} C_DIS
LIN {X 0.088,Y -522.292,Z 1320.914,A 0.000,B 0.000,C 90.000,E1 20.429} C_DIS
LIN {X 0.216,Y -511.846,Z 1320.907,A 0.000,B 0.000,C 90.000,E1 19.322} C_DIS
LIN {X -0.027,Y -502.716,Z 1320.902,A 0.000,B 0.000,C 90.000,E1 18.417} C_DIS
LIN {X -0.100,Y -491.523,Z 1320.896,A 0.000,B 0.000,C 90.000,E1 17.330} C_DIS
LIN {X -0.124,Y -483.372,Z 1320.892,A 0.000,B 0.000,C 90.000,E1 16.551} C_DIS
LIN {X 0.093,Y -473.533,Z 1320.887,A 0.000,B 0.000,C 90.000,E1 15.607} C_DIS
LIN {X -0.037,Y -460.371,Z 1320.880,A 0.000,B 0.000,C 90.000,E1 14.411} C_DIS
LIN {X 0.100,Y -435.826,Z 1320.867,A 0.000,B 0.000,C 90.000,E1 12.007} C_DIS
LIN {X 0.004,Y -418.668,Z 1320.857,A 0.000,B 0.000,C 90.000,E1 10.197} C_DIS
LIN {X -0.022,Y -404.435,Z 1320.848,A 0.000,B 0.000,C 90.000,E1 8.624} C_DIS
LIN {X -0.141,Y -398.667,Z 1320.844,A 0.000,B 0.000,C 90.000,E1 7.992} C_DIS
LIN {X 0.124,Y -395.414,Z 1320.842,A 0.000,B 0.000,C 90.000,E1 7.473} C_DIS
LIN {X 0.089,Y -395.383,Z 1320.842,A 0.000,B 0.000,C 90.000,E1 7.473} C_DIS
LIN {X 0.165,Y -396.138,Z 1320.841,A 0.000,B 0.000,C 90.000,E1 7.296} C_DIS
LIN {X 0.127,Y -396.194,Z 1320.841,A 0.000,B 0.000,C 90.000,E1 7.296} C_DIS
LIN {X 0.021,Y -398.921,Z 1320.839,A 0.000,B 0.000,C 90.000,E1 7.068} C_DIS
LIN {X 0.113,Y -404.304,Z 1320.837,A 0.000,B 0.000,C 90.000,E1 6.663} C_DIS
LIN {X -0.137,Y -412.284,Z 1320.834,A 0.000,B 0.000,C 90.000,E1 6.201} C_DIS
LIN {X 0.006,Y -417.285,Z 1320.833,A 0.000,B 0.000,C 90.000,E1 5.853} C_DIS
LIN {X -0.037,Y -425.169,Z 1320.829,A 0.000,B 0.000,C 90.000,E1 5.277} C_DIS
LIN {X 0.196,Y -429.920,Z 1320.827,A 0.000,B 0.000,C 90.000,E1 4.878} C_DIS
LIN {X -0.105,Y -438.845,Z 1320.823,A 0.000,B 0.000,C 90.000,E1 4.131} C_DIS
LIN {X 0.039,Y -441.912,Z 1320.821,A 0.000,B 0.000,C 90.000,E1 3.841} C_DIS
LIN {X 0.142,Y -450.601,Z 1320.817,A 0.000,B 0.000,C 90.000,E1 2.980} C_DIS
LIN {X -0.099,Y -454.907,Z 1320.814,A 0.000,B 0.000,C 90.000,E1 2.579} C_DIS
LIN {X -0.087,Y -461.688,Z 1320.810,A 0.000,B 0.000,C 90.000,E1 1.835} C_DIS
LIN {X 0.201,Y -468.257,Z 1320.806,A 0.000,B 0.000,C 90.000,E1 1.031} C_DIS
LIN {X -0.012,Y -475.469,Z 1320.801,A 0.000,B 0.000,C 90.000,E1 0.115} C_DIS
LIN {X 0.117,Y -480.900,Z 1320.796,A 0.000,B 0.000,C 90.000,E1 359.312} C_DIS
LIN {X -0.114,Y -485.863,Z 1320.792,A 0.000,B 0.000,C 90.000,E1 358.568} C_DIS
LIN {X 0.203,Y -490.448,Z 1320.788,A 0.000,B 0.000,C 90.000,E1 357.764} C_DIS
LIN {X 0.055,Y -494.713,Z 1320.784,A 0.000,B 0.000,C 90.000,E1 357.020} C_DIS
LIN {X -0.210,Y -497.905,Z 1320.780,A 0.000,B 0.000,C 90.000,E1 356.445} C_DIS
LIN {X -0.080,Y -502.320,Z 1320.775,A 0.000,B 0.000,C 90.000,E1 355.527} C_DIS
LIN {X -0.094,Y -505.801,Z 1320.771,A 0.000,B 0.000,C 90.000,E1 354.780} C_DIS
LIN {X 0.229,Y -508.349,Z 1320.768,A 0.000,B 0.000,C 90.000,E1 354.147} C_DIS
LIN {X -0.184,Y -511.394,Z 1320.764,A 0.000,B 0.000,C 90.000,E1 353.451} C_DIS
LIN {X 0.181,Y -513.641,Z 1320.760,A 0.000,B 0.000,C 90.000,E1 352.818} C_DIS
LIN {X 0.024,Y -516.751,Z 1320.755,A 0.000,B 0.000,C 90.000,E1 351.951} C_DIS
LIN {X -0.101,Y -519.601,Z 1320.750,A 0.000,B 0.000,C 90.000,E1 351.084} C_DIS
LIN {X -0.200,Y -522.948,Z 1320.744,A 0.000,B 0.000,C 90.000,E1 349.926} C_DIS
LIN {X -0.175,Y -525.161,Z 1320.739,A 0.000,B 0.000,C 90.000,E1 349.050} C_DIS
LIN {X -0.124,Y -527.185,Z 1320.734,A 0.000,B 0.000,C 90.000,E1 348.173} C_DIS
LIN {X 0.094,Y -529.486,Z 1320.728,A 0.000,B 0.000,C 90.000,E1 346.992} C_DIS
LIN {X -0.291,Y -531.320,Z 1320.721,A 0.000,B 0.000,C 90.000,E1 345.880} C_DIS
LIN {X -0.050,Y -532.527,Z 1320.717,A 0.000,B 0.000,C 90.000,E1 344.991} C_DIS
LIN {X 0.205,Y -533.448,Z 1320.712,A 0.000,B 0.000,C 90.000,E1 344.102} C_DIS
LIN {X 0.147,Y -534.233,Z 1320.705,A 0.000,B 0.000,C 90.000,E1 342.960} C_DIS
LIN {X -0.096,Y -534.584,Z 1320.701,A 0.000,B 0.000,C 90.000,E1 342.127} C_DIS
LIN {X -0.171,Y -534.608,Z 1320.696,A 0.000,B 0.000,C 90.000,E1 341.275} C_DIS
LIN {X -0.039,Y -534.135,Z 1320.690,A 0.000,B 0.000,C 90.000,E1 340.115} C_DIS
LIN {X -0.113,Y -533.519,Z 1320.685,A 0.000,B 0.000,C 90.000,E1 339.263} C_DIS
LIN {X -0.001,Y -532.104,Z 1320.678,A 0.000,B 0.000,C 90.000,E1 338.103} C_DIS
LIN {X -0.204,Y -530.155,Z 1320.672,A 0.000,B 0.000,C 90.000,E1 336.975} C_DIS
LIN {X -0.014,Y -529.487,Z 1320.670,A 0.000,B 0.000,C 90.000,E1 336.666} C_DIS
LIN {X -0.127,Y -528.380,Z 1320.667,A 0.000,B 0.000,C 90.000,E1 336.102} C_DIS
LIN {X -0.073,Y -526.091,Z 1320.662,A 0.000,B 0.000,C 90.000,E1 335.229} C_DIS
LIN {X -0.137,Y -522.513,Z 1320.656,A 0.000,B 0.000,C 90.000,E1 334.076} C_DIS
LIN {X 0.215,Y -518.845,Z 1320.649,A 0.000,B 0.000,C 90.000,E1 332.871} C_DIS
LIN {X -0.053,Y -514.142,Z 1320.641,A 0.000,B 0.000,C 90.000,E1 331.435} C_DIS
LIN {X -0.047,Y -510.134,Z 1320.635,A 0.000,B 0.000,C 90.000,E1 330.255} C_DIS
LIN {X 0.264,Y -507.000,Z 1320.630,A 0.000,B 0.000,C 90.000,E1 329.331} C_DIS
LIN {X -0.278,Y -502.410,Z 1320.623,A 0.000,B 0.000,C 90.000,E1 328.201} C_DIS
LIN {X -0.051,Y -495.506,Z 1320.613,A 0.000,B 0.000,C 90.000,E1 326.373} C_DIS
LIN {X 0.098,Y -489.252,Z 1320.604,A 0.000,B 0.000,C 90.000,E1 324.689} C_DIS
LIN {X -0.060,Y -487.846,Z 1320.602,A 0.000,B 0.000,C 90.000,E1 324.402} C_DIS
LIN {X 0.003,Y -487.030,Z 1320.601,A 0.000,B 0.000,C 90.000,E1 324.242} C_DIS
LIN {X 0.172,Y -486.024,Z 1320.601,A 0.000,B 0.000,C 90.000,E1 324.069} C_DIS
LIN {X 0.232,Y -484.482,Z 1320.600,A 0.000,B 0.000,C 90.000,E1 323.909} C_DIS
LIN {X -0.049,Y -462.287,Z 1320.589,A 0.000,B 0.000,C 90.000,E1 321.949} C_DIS
LIN {X 0.047,Y -441.048,Z 1320.577,A 0.000,B 0.000,C 90.000,E1 319.784} C_DIS
LIN {X -0.026,Y -421.854,Z 1320.564,A 0.000,B 0.000,C 90.000,E1 317.595} C_DIS
LIN {X -0.212,Y -403.506,Z 1320.551,A 0.000,B 0.000,C 90.000,E1 315.243} C_DIS
LIN {X -0.145,Y -386.773,Z 1320.538,A 0.000,B 0.000,C 90.000,E1 312.771} C_DIS
LIN {X 0.037,Y -383.122,Z 1320.534,A 0.000,B 0.000,C 90.000,E1 312.162} C_DIS
LIN {X 0.001,Y -383.095,Z 1320.534,A 0.000,B 0.000,C 90.000,E1 312.162} C_DIS
LIN {X 0.057,Y -384.719,Z 1320.528,A 0.000,B 0.000,C 90.000,E1 310.943} C_DIS
LIN {X -0.085,Y -390.400,Z 1320.496,A 0.000,B 0.000,C 90.000,E1 305.231} C_DIS
LIN {X 0.147,Y -391.337,Z 1320.492,A 0.000,B 0.000,C 90.000,E1 304.485} C_DIS
LIN {X -0.030,Y -397.048,Z 1320.458,A 0.000,B 0.000,C 90.000,E1 298.487} C_DIS
LIN {X -0.250,Y -401.433,Z 1320.427,A 0.000,B 0.000,C 90.000,E1 292.898} C_DIS
LIN {X -0.014,Y -401.673,Z 1320.425,A 0.000,B 0.000,C 90.000,E1 292.514} C_DIS
LIN {X 0.116,Y -404.763,Z 1320.394,A 0.000,B 0.000,C 90.000,E1 286.913} C_DIS
LIN {X 0.022,Y -406.154,Z 1320.363,A 0.000,B 0.000,C 90.000,E1 281.366} C_DIS
LIN {X 0.127,Y -405.644,Z 1320.334,A 0.000,B 0.000,C 90.000,E1 276.144} C_DIS
LIN {X 0.132,Y -405.636,Z 1320.332,A 0.000,B 0.000,C 90.000,E1 275.796} C_DIS
LIN {X -0.198,Y -403.556,Z 1320.305,A 0.000,B 0.000,C 90.000,E1 270.974} C_DIS
LIN {X 0.140,Y -403.093,Z 1320.301,A 0.000,B 0.000,C 90.000,E1 270.229} C_DIS
LIN {X -0.034,Y -399.032,Z 1320.272,A 0.000,B 0.000,C 90.000,E1 265.008} C_DIS
LIN {X -0.116,Y -398.171,Z 1320.268,A 0.000,B 0.000,C 90.000,E1 264.318} C_DIS
LIN {X 0.136,Y -392.958,Z 1320.241,A 0.000,B 0.000,C 90.000,E1 259.342} C_DIS
LIN {X 0.094,Y -392.536,Z 1320.239,A 0.000,B 0.000,C 90.000,E1 258.993} C_DIS
LIN {X -0.131,Y -386.160,Z 1320.213,A 0.000,B 0.000,C 90.000,E1 254.393} C_DIS
LIN {X -0.167,Y -385.045,Z 1320.207,A 0.000,B 0.000,C 90.000,E1 253.323} C_DIS
LIN {X 0.073,Y -378.177,Z 1320.183,A 0.000,B 0.000,C 90.000,E1 248.954} C_DIS
LIN {X -0.060,Y -375.949,Z 1320.173,A 0.000,B 0.000,C 90.000,E1 247.155} C_DIS
LIN {X -0.094,Y -369.155,Z 1320.151,A 0.000,B 0.000,C 90.000,E1 243.127} C_DIS
LIN {X -0.185,Y -366.302,Z 1320.138,A 0.000,B 0.000,C 90.000,E1 240.923} C_DIS
LIN {X 0.208,Y -358.390,Z 1320.111,A 0.000,B 0.000,C 90.000,E1 236.008} C_DIS
LIN {X 0.051,Y -356.084,Z 1320.101,A 0.000,B 0.000,C 90.000,E1 234.149} C_DIS
LIN {X -0.107,Y -354.778,Z 1320.097,A 0.000,B 0.000,C 90.000,E1 233.417} C_DIS
LIN {X -0.126,Y -354.779,Z 1320.097,A 0.000,B 0.000,C 90.000,E1 233.417} C_DIS
LIN {X -0.193,Y -368.070,Z 1320.082,A 0.000,B 0.000,C 90.000,E1 230.803} C_DIS
LIN {X -0.243,Y -382.870,Z 1320.068,A 0.000,B 0.000,C 90.000,E1 228.243} C_DIS
LIN {X -0.163,Y -399.262,Z 1320.054,A 0.000,B 0.000,C 90.000,E1 225.729} C_DIS
LIN {X -0.169,Y -417.371,Z 1320.041,A 0.000,B 0.000,C 90.000,E1 223.299} C_DIS
LIN {X -0.018,Y -436.736,Z 1320.028,A 0.000,B 0.000,C 90.000,E1 220.987} C_DIS
LIN {X -0.090,Y -442.392,Z 1320.024,A 0.000,B 0.000,C 90.000,E1 220.378} C_DIS
LIN {X -0.014,Y -443.530,Z 1320.023,A 0.000,B 0.000,C 90.000,E1 220.216} C_DIS
LIN {X -0.225,Y -444.296,Z 1320.023,A 0.000,B 0.000,C 90.000,E1 220.092} C_DIS
LIN {X 0.085,Y -445.484,Z 1320.021,A 0.000,B 0.000,C 90.000,E1 219.725} C_DIS
LIN {X 0.056,Y -446.373,Z 1320.019,A 0.000,B 0.000,C 90.000,E1 219.402} C_DIS
LIN {X 0.070,Y -447.737,Z 1320.015,A 0.000,B 0.000,C 90.000,E1 218.749} C_DIS
LIN {X 0.096,Y -448.773,Z 1320.012,A 0.000,B 0.000,C 90.000,E1 218.096} C_DIS
LIN {X -0.163,Y -449.897,Z 1320.006,A 0.000,B 0.000,C 90.000,E1 217.156} C_DIS
LIN {X 0.004,Y -451.296,Z 1319.997,A 0.000,B 0.000,C 90.000,E1 215.518} C_DIS
LIN {X 0.022,Y -454.459,Z 1319.979,A 0.000,B 0.000,C 90.000,E1 212.291} C_DIS
LIN {X -0.033,Y -456.989,Z 1319.967,A 0.000,B 0.000,C 90.000,E1 210.050} C_DIS
LIN {X 0.193,Y -459.383,Z 1319.956,A 0.000,B 0.000,C 90.000,E1 208.103} C_DIS
LIN {X -0.100,Y -462.988,Z 1319.942,A 0.000,B 0.000,C 90.000,E1 205.591} C_DIS
LIN {X -0.077,Y -465.313,Z 1319.933,A 0.000,B 0.000,C 90.000,E1 204.003} C_DIS
LIN {X 0.103,Y -467.092,Z 1319.926,A 0.000,B 0.000,C 90.000,E1 202.717} C_DIS
LIN {X 0.113,Y -468.419,Z 1319.921,A 0.000,B 0.000,C 90.000,E1 201.770} C_DIS
LIN {X 0.008,Y -471.745,Z 1319.907,A 0.000,B 0.000,C 90.000,E1 199.268} C_DIS
LIN {X -0.119,Y -474.747,Z 1319.895,A 0.000,B 0.000,C 90.000,E1 197.094} C_DIS
LIN {X -0.121,Y -476.846,Z 1319.886,A 0.000,B 0.000,C 90.000,E1 195.536} C_DIS
LIN {X 0.095,Y -479.250,Z 1319.876,A 0.000,B 0.000,C 90.000,E1 193.647} C_DIS
LIN {X -0.209,Y -481.647,Z 1319.866,A 0.000,B 0.000,C 90.000,E1 191.827} C_DIS
LIN {X -0.085,Y -484.058,Z 1319.855,A 0.000,B 0.000,C 90.000,E1 189.962} C_DIS
LIN {X -0.112,Y -486.796,Z 1319.843,A 0.000,B 0.000,C 90.000,E1 187.814} C_DIS
LIN {X 0.103,Y -488.578,Z 1319.835,A 0.000,B 0.000,C 90.000,E1 186.258} C_DIS
LIN {X -0.136,Y -490.221,Z 1319.826,A 0.000,B 0.000,C 90.000,E1 184.759} C_DIS
LIN {X 0.225,Y -491.323,Z 1319.820,A 0.000,B 0.000,C 90.000,E1 183.498} C_DIS
LIN {X -0.032,Y -492.558,Z 1319.811,A 0.000,B 0.000,C 90.000,E1 182.007} C_DIS
LIN {X -0.125,Y -493.302,Z 1319.804,A 0.000,B 0.000,C 90.000,E1 180.802} C_DIS
LIN {X -0.216,Y -493.875,Z 1319.798,A 0.000,B 0.000,C 90.000,E1 179.599} C_DIS
LIN {X -0.158,Y -494.153,Z 1319.793,A 0.000,B 0.000,C 90.000,E1 178.682} C_DIS
LIN {X -0.227,Y -494.220,Z 1319.786,A 0.000,B 0.000,C 90.000,E1 177.478} C_DIS
LIN {X 0.199,Y -494.006,Z 1319.779,A 0.000,B 0.000,C 90.000,E1 176.216} C_DIS
LIN {X -0.218,Y -493.538,Z 1319.774,A 0.000,B 0.000,C 90.000,E1 175.355} C_DIS
LIN {X 0.226,Y -492.682,Z 1319.767,A 0.000,B 0.000,C 90.000,E1 174.090} C_DIS
LIN {X -0.157,Y -491.802,Z 1319.762,A 0.000,B 0.000,C 90.000,E1 173.223} C_DIS
LIN {X -0.059,Y -490.651,Z 1319.757,A 0.000,B 0.000,C 90.000,E1 172.299} C_DIS
LIN {X 0.025,Y -489.180,Z 1319.752,A 0.000,B 0.000,C 90.000,E1 171.376} C_DIS
LIN {X -0.202,Y -488.048,Z 1319.749,A 0.000,B 0.000,C 90.000,E1 170.792} C_DIS
LIN {X 0.047,Y -486.798,Z 1319.745,A 0.000,B 0.000,C 90.000,E1 170.151} C_DIS
LIN {X -0.189,Y -485.382,Z 1319.742,A 0.000,B 0.000,C 90.000,E1 169.567} C_DIS
LIN {X -0.086,Y -482.958,Z 1319.737,A 0.000,B 0.000,C 90.000,E1 168.634} C_DIS
LIN {X -0.156,Y -478.652,Z 1319.730,A 0.000,B 0.000,C 90.000,E1 167.409} C_DIS
LIN {X 0.164,Y -477.346,Z 1319.728,A 0.000,B 0.000,C 90.000,E1 167.061} C_DIS
LIN {X 0.055,Y -473.464,Z 1319.724,A 0.000,B 0.000,C 90.000,E1 166.297} C_DIS
LIN {X -0.154,Y -467.008,Z 1319.718,A 0.000,B 0.000,C 90.000,E1 165.227} C_DIS
LIN {X 0.127,Y -456.537,Z 1319.708,A 0.000,B 0.000,C 90.000,E1 163.449} C_DIS
LIN {X -0.011,Y -449.408,Z 1319.701,A 0.000,B 0.000,C 90.000,E1 162.181} C_DIS
LIN {X -0.251,Y -445.689,Z 1319.697,A 0.000,B 0.000,C 90.000,E1 161.402} C_DIS
LIN {X 0.039,Y -443.180,Z 1319.692,A 0.000,B 0.000,C 90.000,E1 160.550} C_DIS
LIN {X -0.187,Y -443.102,Z 1319.689,A 0.000,B 0.000,C 90.000,E1 160.061} C_DIS
LIN {X -0.051,Y -443.201,Z 1319.688,A 0.000,B 0.000,C 90.000,E1 159.880} C_DIS
LIN {X -0.019,Y -444.001,Z 1319.687,A 0.000,B 0.000,C 90.000,E1 159.625} C_DIS
LIN {X -0.059,Y -444.042,Z 1319.687,A 0.000,B 0.000,C 90.000,E1 159.625} C_DIS
LIN {X -0.180,Y -446.387,Z 1319.685,A 0.000,B 0.000,C 90.000,E1 159.390} C_DIS
LIN {X -0.010,Y -448.051,Z 1319.684,A 0.000,B 0.000,C 90.000,E1 159.135} C_DIS
LIN {X 0.102,Y -452.057,Z 1319.682,A 0.000,B 0.000,C 90.000,E1 158.773} C_DIS
LIN {X -0.042,Y -470.125,Z 1319.674,A 0.000,B 0.000,C 90.000,E1 157.358} C_DIS
LIN {X -0.162,Y -479.093,Z 1319.670,A 0.000,B 0.000,C 90.000,E1 156.666} C_DIS
LIN {X -0.224,Y -488.140,Z 1319.666,A 0.000,B 0.000,C 90.000,E1 155.921} C_DIS
LIN {X 0.132,Y -495.230,Z 1319.662,A 0.000,B 0.000,C 90.000,E1 155.229} C_DIS
LIN {X -0.197,Y -502.137,Z 1319.659,A 0.000,B 0.000,C 90.000,E1 154.588} C_DIS
LIN {X -0.057,Y -506.256,Z 1319.656,A 0.000,B 0.000,C 90.000,E1 154.152} C_DIS
LIN {X 0.259,Y -513.961,Z 1319.652,A 0.000,B 0.000,C 90.000,E1 153.256} C_DIS
LIN {X -0.200,Y -517.608,Z 1319.649,A 0.000,B 0.000,C 90.000,E1 152.871} C_DIS
LIN {X 0.161,Y -519.990,Z 1319.648,A 0.000,B 0.000,C 90.000,E1 152.538} C_DIS
LIN {X -0.035,Y -524.178,Z 1319.644,A 0.000,B 0.000,C 90.000,E1 151.975} C_DIS
LIN {X 0.043,Y -527.913,Z 1319.641,A 0.000,B 0.000,C 90.000,E1 151.385} C_DIS
LIN {X 0.000,Y -531.740,Z 1319.637,A 0.000,B 0.000,C 90.000,E1 150.667} C_DIS
LIN {X -0.014,Y -534.697,Z 1319.633,A 0.000,B 0.000,C 90.000,E1 149.950} C_DIS
LIN {X -0.326,Y -536.704,Z 1319.630,A 0.000,B 0.000,C 90.000,E1 149.410} C_DIS
LIN {X -0.164,Y -539.114,Z 1319.625,A 0.000,B 0.000,C 90.000,E1 148.535} C_DIS
LIN {X 0.026,Y -541.040,Z 1319.620,A 0.000,B 0.000,C 90.000,E1 147.661} C_DIS
LIN {X -0.218,Y -542.566,Z 1319.616,A 0.000,B 0.000,C 90.000,E1 146.834} C_DIS
LIN {X 0.282,Y -543.457,Z 1319.613,A 0.000,B 0.000,C 90.000,E1 146.215} C_DIS
LIN {X 0.134,Y -545.179,Z 1319.605,A 0.000,B 0.000,C 90.000,E1 144.815} C_DIS
LIN {X 0.012,Y -546.575,Z 1319.597,A 0.000,B 0.000,C 90.000,E1 143.417} C_DIS
LIN {X 0.043,Y -547.796,Z 1319.590,A 0.000,B 0.000,C 90.000,E1 142.145} C_DIS
LIN {X -0.089,Y -548.408,Z 1319.588,A 0.000,B 0.000,C 90.000,E1 141.823} C_DIS
LIN {X 0.051,Y -548.809,Z 1319.586,A 0.000,B 0.000,C 90.000,E1 141.492} C_DIS
LIN {X -0.217,Y -549.730,Z 1319.585,A 0.000,B 0.000,C 90.000,E1 141.331} C_DIS
LIN {X 0.085,Y -549.783,Z 1319.585,A 0.000,B 0.000,C 90.000,E1 141.295} C_DIS
LIN {X -0.245,Y -553.905,Z 1319.584,A 0.000,B 0.000,C 90.000,E1 141.090} C_DIS
LIN {X 0.161,Y -566.717,Z 1319.582,A 0.000,B 0.000,C 90.000,E1 140.642} C_DIS
LIN {X -0.213,Y -572.474,Z 1319.580,A 0.000,B 0.000,C 90.000,E1 140.436} C_DIS
LIN {X -0.119,Y -578.511,Z 1319.578,A 0.000,B 0.000,C 90.000,E1 140.114} C_DIS
LIN {X -0.096,Y -584.303,Z 1319.576,A 0.000,B 0.000,C 90.000,E1 139.747} C_DIS
LIN {X 0.162,Y -589.799,Z 1319.574,A 0.000,B 0.000,C 90.000,E1 139.299} C_DIS
LIN {X -0.080,Y -592.472,Z 1319.573,A 0.000,B 0.000,C 90.000,E1 139.094} C_DIS
LIN {X 0.331,Y -593.827,Z 1319.572,A 0.000,B 0.000,C 90.000,E1 138.933} C_DIS
LIN {X -0.097,Y -595.409,Z 1319.571,A 0.000,B 0.000,C 90.000,E1 138.852} C_DIS
LIN {X 0.093,Y -600.062,Z 1319.569,A 0.000,B 0.000,C 90.000,E1 138.405} C_DIS
LIN {X -0.013,Y -603.644,Z 1319.567,A 0.000,B 0.000,C 90.000,E1 138.038} C_DIS
LIN {X 0.194,Y -607.152,Z 1319.565,A 0.000,B 0.000,C 90.000,E1 137.634} C_DIS
LIN {X -0.188,Y -611.513,Z 1319.562,A 0.000,B 0.000,C 90.000,E1 137.148} C_DIS
LIN {X -0.095,Y -615.606,Z 1319.559,A 0.000,B 0.000,C 90.000,E1 136.620} C_DIS
LIN {X 0.007,Y -619.494,Z 1319.556,A 0.000,B 0.000,C 90.000,E1 136.095} C_DIS
LIN {X 0.013,Y -624.775,Z 1319.552,A 0.000,B 0.000,C 90.000,E1 135.324} C_DIS
LIN {X 0.005,Y -630.618,Z 1319.547,A 0.000,B 0.000,C 90.000,E1 134.433} C_DIS
LIN {X -0.226,Y -633.842,Z 1319.544,A 0.000,B 0.000,C 90.000,E1 133.947} C_DIS
LIN {X 0.240,Y -640.695,Z 1319.538,A 0.000,B 0.000,C 90.000,E1 132.771} C_DIS
LIN {X -0.106,Y -648.005,Z 1319.531,A 0.000,B 0.000,C 90.000,E1 131.553} C_DIS
LIN {X -0.290,Y -653.002,Z 1319.526,A 0.000,B 0.000,C 90.000,E1 130.701} C_DIS
LIN {X 0.076,Y -657.813,Z 1319.521,A 0.000,B 0.000,C 90.000,E1 129.806} C_DIS
LIN {X 0.126,Y -662.890,Z 1319.516,A 0.000,B 0.000,C 90.000,E1 128.830} C_DIS
LIN {X -0.287,Y -667.580,Z 1319.510,A 0.000,B 0.000,C 90.000,E1 127.890} C_DIS
LIN {X 0.200,Y -669.759,Z 1319.508,A 0.000,B 0.000,C 90.000,E1 127.363} C_DIS
LIN {X 0.295,Y -671.848,Z 1319.505,A 0.000,B 0.000,C 90.000,E1 126.870} C_DIS
LIN {X -0.015,Y -675.583,Z 1319.500,A 0.000,B 0.000,C 90.000,E1 125.931} C_DIS
LIN {X -0.122,Y -678.919,Z 1319.494,A 0.000,B 0.000,C 90.000,E1 124.978} C_DIS
LIN {X 0.033,Y -681.133,Z 1319.490,A 0.000,B 0.000,C 90.000,E1 124.246} C_DIS
LIN {X 0.002,Y -683.695,Z 1319.485,A 0.000,B 0.000,C 90.000,E1 123.293} C_DIS
LIN {X 0.385,Y -685.399,Z 1319.481,A 0.000,B 0.000,C 90.000,E1 122.546} C_DIS
LIN {X -0.160,Y -686.920,Z 1319.477,A 0.000,B 0.000,C 90.000,E1 121.878} C_DIS
LIN {X -0.116,Y -688.673,Z 1319.472,A 0.000,B 0.000,C 90.000,E1 120.924} C_DIS
LIN {X -0.038,Y -689.776,Z 1319.468,A 0.000,B 0.000,C 90.000,E1 120.207} C_DIS
LIN {X -0.310,Y -691.046,Z 1319.463,A 0.000,B 0.000,C 90.000,E1 119.283} C_DIS
LIN {X 0.039,Y -691.714,Z 1319.457,A 0.000,B 0.000,C 90.000,E1 118.309} C_DIS
LIN {X 0.155,Y -692.059,Z 1319.453,A 0.000,B 0.000,C 90.000,E1 117.590} C_DIS
LIN {X -0.105,Y -692.240,Z 1319.448,A 0.000,B 0.000,C 90.000,E1 116.668} C_DIS
LIN {X 0.074,Y -692.224,Z 1319.446,A 0.000,B 0.000,C 90.000,E1 116.181} C_DIS
LIN {X 0.183,Y -691.831,Z 1319.442,A 0.000,B 0.000,C 90.000,E1 115.463} C_DIS
LIN {X -0.254,Y -691.409,Z 1319.439,A 0.000,B 0.000,C 90.000,E1 115.027} C_DIS
LIN {X 0.225,Y -690.740,Z 1319.436,A 0.000,B 0.000,C 90.000,E1 114.515} C_DIS
LIN {X -0.216,Y -689.440,Z 1319.434,A 0.000,B 0.000,C 90.000,E1 114.079} C_DIS
LIN {X 0.016,Y -688.632,Z 1319.432,A 0.000,B 0.000,C 90.000,E1 113.823} C_DIS
LIN {X 0.223,Y -686.154,Z 1319.430,A 0.000,B 0.000,C 90.000,E1 113.334} C_DIS
LIN {X 0.334,Y -685.363,Z 1319.429,A 0.000,B 0.000,C 90.000,E1 113.206} C_DIS
LIN {X -0.075,Y -682.825,Z 1319.428,A 0.000,B 0.000,C 90.000,E1 113.003} C_DIS
LIN {X -0.061,Y -680.317,Z 1319.427,A 0.000,B 0.000,C 90.000,E1 112.770} C_DIS
LIN {X 0.107,Y -678.887,Z 1319.426,A 0.000,B 0.000,C 90.000,E1 112.642} C_DIS
LIN {X 0.356,Y -676.731,Z 1319.425,A 0.000,B 0.000,C 90.000,E1 112.514} C_DIS
LIN {X -0.278,Y -674.039,Z 1319.425,A 0.000,B 0.000,C 90.000,E1 112.461} C_DIS
LIN {X -0.186,Y -668.557,Z 1319.424,A 0.000,B 0.000,C 90.000,E1 112.259} C_DIS
LIN {X -0.297,Y -664.413,Z 1319.423,A 0.000,B 0.000,C 90.000,E1 112.153} C_DIS
LIN {X -0.069,Y -657.191,Z 1319.422,A 0.000,B 0.000,C 90.000,E1 112.025} C_DIS
LIN {X 0.363,Y -647.394,Z 1319.422,A 0.000,B 0.000,C 90.000,E1 111.897} C_DIS
LIN {X -0.056,Y -644.154,Z 1319.422,A 0.000,B 0.000,C 90.000,E1 111.897} C_DIS
LIN {X -0.197,Y -642.130,Z 1319.421,A 0.000,B 0.000,C 90.000,E1 111.844} C_DIS
LIN {X -0.259,Y -642.149,Z 1319.421,A 0.000,B 0.000,C 90.000,E1 111.844} C_DIS
LIN {X 0.186,Y -642.888,Z 1319.421,A 0.000,B 0.000,C 90.000,E1 111.663} C_DIS
LIN {X 0.166,Y -644.867,Z 1319.419,A 0.000,B 0.000,C 90.000,E1 111.408} C_DIS
LIN {X 0.030,Y -647.906,Z 1319.417,A 0.000,B 0.000,C 90.000,E1 111.046} C_DIS
LIN {X -0.049,Y -651.730,Z 1319.414,A 0.000,B 0.000,C 90.000,E1 110.556} C_DIS
LIN {X -0.060,Y -655.940,Z 1319.411,A 0.000,B 0.000,C 90.000,E1 109.939} C_DIS
LIN {X -0.039,Y -659.614,Z 1319.407,A 0.000,B 0.000,C 90.000,E1 109.322} C_DIS
LIN {X -0.209,Y -662.717,Z 1319.404,A 0.000,B 0.000,C 90.000,E1 108.725} C_DIS
LIN {X -0.297,Y -665.964,Z 1319.400,A 0.000,B 0.000,C 90.000,E1 108.000} C_DIS
LIN {X 0.283,Y -668.760,Z 1319.396,A 0.000,B 0.000,C 90.000,E1 107.221} C_DIS
LIN {X 0.252,Y -671.224,Z 1319.392,A 0.000,B 0.000,C 90.000,E1 106.496} C_DIS
LIN {X 0.117,Y -672.748,Z 1319.389,A 0.000,B 0.000,C 90.000,E1 106.024} C_DIS
LIN {X 0.115,Y -674.561,Z 1319.385,A 0.000,B 0.000,C 90.000,E1 105.300} C_DIS
LIN {X -0.051,Y -676.085,Z 1319.381,A 0.000,B 0.000,C 90.000,E1 104.592} C_DIS
LIN {X -0.199,Y -677.377,Z 1319.377,A 0.000,B 0.000,C 90.000,E1 103.883} C_DIS
LIN {X 0.322,Y -678.291,Z 1319.373,A 0.000,B 0.000,C 90.000,E1 103.119} C_DIS
LIN {X 0.192,Y -678.682,Z 1319.369,A 0.000,B 0.000,C 90.000,E1 102.411} C_DIS
LIN {X -0.036,Y -678.824,Z 1319.366,A 0.000,B 0.000,C 90.000,E1 101.951} C_DIS
LIN {X -0.121,Y -678.796,Z 1319.364,A 0.000,B 0.000,C 90.000,E1 101.478} C_DIS
END
